LIN {X 0,Y 247.76,Z 536.952,A -85,B 0,C 180,E1 -18799.376,E2 -18799.376} C_VEL
LIN {X 0,Y 247.256,Z 541.833,A -85,B 0,C 180,E1 -18801.831,E2 -18801.831} C_VEL
LIN {X 0,Y 246.931,Z 545.565,A -85,B 0,C 180,E1 -18804.284,E2 -18804.284} C_VEL
LIN {X 0,Y 246.895,Z 548.265,A -85,B 0,C 180,E1 -18806.738,E2 -18806.738} C_VEL
LIN {X 0,Y 246.957,Z 549.533,A -85,B 0,C 180,E1 -18808.37,E2 -18808.37} C_VEL
LIN {X 0,Y 246.985,Z 550.397,A -85,B 0,C 180,E1 -18810.001,E2 -18810.001} C_VEL
LIN {X 0,Y 246.925,Z 550.819,A -85,B 0,C 180,E1 -18811.632,E2 -18811.632} C_VEL
LIN {X 0,Y 246.882,Z 550.489,A -85,B 0,C 180,E1 -18814.9,E2 -18814.9} C_VEL
LIN {X 0,Y 247.022,Z 549.754,A -85,B 0,C 180,E1 -18816.536,E2 -18816.536} C_VEL
LIN {X 0,Y 247.296,Z 548.597,A -85,B 0,C 180,E1 -18818.17,E2 -18818.17} C_VEL
LIN {X 0,Y 247.735,Z 547.02,A -85,B 0,C 180,E1 -18819.801,E2 -18819.801} C_VEL
LIN {X 0,Y 248.65,Z 543.875,A -85,B 0,C 180,E1 -18822.24,E2 -18822.24} C_VEL
LIN {X 0,Y 249.943,Z 539.694,A -85,B 0,C 180,E1 -18824.66,E2 -18824.66} C_VEL
LIN {X 0,Y 252.206,Z 533.352,A -85,B 0,C 180,E1 -18827.432,E2 -18827.432} C_VEL
LIN {X 0,Y 254.652,Z 525.61,A -85,B 0,C 180,E1 -18830.038,E2 -18830.038} C_VEL
LIN {X 0,Y 256.959,Z 517.893,A -85,B 0,C 180,E1 -18832.092,E2 -18832.092} C_VEL
LIN {X 0,Y 259.561,Z 509.116,A -85,B 0,C 180,E1 -18833.964,E2 -18833.964} C_VEL
LIN {X 0,Y 262.449,Z 498.336,A -85,B 0,C 180,E1 -18835.796,E2 -18835.796} C_VEL
LIN {X 0,Y 264.991,Z 487.513,A -85,B 0,C 180,E1 -18837.227,E2 -18837.227} C_VEL
LIN {X 0,Y 267.415,Z 475.396,A -85,B 0,C 180,E1 -18838.448,E2 -18838.448} C_VEL
LIN {X 0,Y 269.44,Z 462.72,A -85,B 0,C 180,E1 -18839.388,E2 -18839.388} C_VEL
LIN {X 0,Y 270.794,Z 450.762,A -85,B 0,C 180,E1 -18839.998,E2 -18839.998} C_VEL
LIN {X 0,Y 271.642,Z 434.886,A -85,B 0,C 180,E1 -18840.499,E2 -18840.499} C_VEL
LIN {X 0,Y 273.321,Z 390.073,A -85,B 0,C 180,E1 -18841.676,E2 -18841.676} C_VEL
LIN {X 0,Y 270.28,Z 372.943,A -85,B 0,C 180,E1 -18842.701,E2 -18842.701} C_VEL
LIN {X 0,Y 265.11,Z 361.26,A -85,B 0,C 180,E1 -18843.938,E2 -18843.938} C_VEL
LIN {X 0,Y 257.601,Z 346.459,A -85,B 0,C 180,E1 -18845.793,E2 -18845.793} C_VEL
LIN {X 0,Y 254.306,Z 340.666,A -85,B 0,C 180,E1 -18846.634,E2 -18846.634} C_VEL
LIN {X 0,Y 252.61,Z 337.257,A -85,B 0,C 180,E1 -18847.12,E2 -18847.12} C_VEL
LIN {X 0,Y 250.483,Z 329.649,A -85,B 0,C 180,E1 -18850.751,E2 -18850.751} C_VEL
LIN {X 0,Y 249.027,Z 324.462,A -85,B 0,C 180,E1 -18853.427,E2 -18853.427} C_VEL
LIN {X 0,Y 249.012,Z 324.468,A -85,B 0,C 180,E1 -18857.362,E2 -18857.362} C_VEL
LIN {X 0,Y 249.027,Z 324.458,A -85,B 0,C 180,E1 -18861.62,E2 -18861.62} C_VEL
LIN {X 0,Y 249.045,Z 324.46,A -85,B 0,C 180,E1 -18865.64,E2 -18865.64} C_VEL
LIN {X 0,Y 249.005,Z 324.468,A -85,B 0,C 180,E1 -18869.467,E2 -18869.467} C_VEL
LIN {X 0,Y 249.04,Z 324.464,A -85,B 0,C 180,E1 -18873.159,E2 -18873.159} C_VEL
LIN {X 0,Y 249.128,Z 324.445,A -85,B 0,C 180,E1 -18874.966,E2 -18874.966} C_VEL
LIN {X 0,Y 249.092,Z 324.45,A -85,B 0,C 180,E1 -18878.605,E2 -18878.605} C_VEL
LIN {X 0,Y 249.179,Z 324.436,A -85,B 0,C 180,E1 -18883.618,E2 -18883.618} C_VEL
LIN {X 0,Y 249.237,Z 324.432,A -85,B 0,C 180,E1 -18888.616,E2 -18888.616} C_VEL
LIN {X 0,Y 249.448,Z 324.398,A -85,B 0,C 180,E1 -18891.902,E2 -18891.902} C_VEL
LIN {X 0,Y 249.281,Z 324.423,A -85,B 0,C 180,E1 -18895.148,E2 -18895.148} C_VEL
LIN {X 0,Y 249.666,Z 324.381,A -85,B 0,C 180,E1 -18898.387,E2 -18898.387} C_VEL
LIN {X 0,Y 249.673,Z 324.375,A -85,B 0,C 180,E1 -18901.613,E2 -18901.613} C_VEL
LIN {X 0,Y 249.432,Z 324.41,A -85,B 0,C 180,E1 -18906.577,E2 -18906.577} C_VEL
LIN {X 0,Y 249.346,Z 324.415,A -85,B 0,C 180,E1 -18909.737,E2 -18909.737} C_VEL
LIN {X 0,Y 249.185,Z 324.441,A -85,B 0,C 180,E1 -18914.705,E2 -18914.705} C_VEL
LIN {X 0,Y 249.116,Z 324.444,A -85,B 0,C 180,E1 -18918.08,E2 -18918.08} C_VEL
LIN {X 0,Y 249.084,Z 324.447,A -85,B 0,C 180,E1 -18921.519,E2 -18921.519} C_VEL
LIN {X 0,Y 249.108,Z 324.445,A -85,B 0,C 180,E1 -18925.469,E2 -18925.469} C_VEL
LIN {X 0,Y 249.045,Z 324.454,A -85,B 0,C 180,E1 -18928.976,E2 -18928.976} C_VEL
LIN {X 0,Y 249.031,Z 324.459,A -85,B 0,C 180,E1 -18932.426,E2 -18932.426} C_VEL
LIN {X 0,Y 249.057,Z 324.462,A -85,B 0,C 180,E1 -18936.341,E2 -18936.341} C_VEL
LIN {X 0,Y 249.034,Z 324.542,A -85,B 0,C 180,E1 -18940.134,E2 -18940.134} C_VEL
LIN {X 0,Y 249.7,Z 326.855,A -85,B 0,C 180,E1 -18941.342,E2 -18941.342} C_VEL
LIN {X 0,Y 251.823,Z 330.474,A -85,B 0,C 180,E1 -18941.918,E2 -18941.918} C_VEL
LIN {X 0,Y 258.717,Z 342.019,A -85,B 0,C 180,E1 -18943.683,E2 -18943.683} C_VEL
LIN {X 0,Y 265.785,Z 354.94,A -85,B 0,C 180,E1 -18945.389,E2 -18945.389} C_VEL
LIN {X 0,Y 272.354,Z 368.856,A -85,B 0,C 180,E1 -18946.92,E2 -18946.92} C_VEL
LIN {X 0,Y 274.083,Z 372.882,A -85,B 0,C 180,E1 -18947.317,E2 -18947.317} C_VEL
LIN {X 0,Y 271.457,Z 434.189,A -85,B 0,C 180,E1 -18948.929,E2 -18948.929} C_VEL
LIN {X 0,Y 270.158,Z 447.569,A -85,B 0,C 180,E1 -18949.553,E2 -18949.553} C_VEL
LIN {X 0,Y 268.442,Z 460.42,A -85,B 0,C 180,E1 -18950.466,E2 -18950.466} C_VEL
LIN {X 0,Y 266.639,Z 470.957,A -85,B 0,C 180,E1 -18951.485,E2 -18951.485} C_VEL
LIN {X 0,Y 264.44,Z 481.999,A -85,B 0,C 180,E1 -18952.875,E2 -18952.875} C_VEL
LIN {X 0,Y 261.843,Z 492.45,A -85,B 0,C 180,E1 -18954.519,E2 -18954.519} C_VEL
LIN {X 0,Y 259.378,Z 501.292,A -85,B 0,C 180,E1 -18956.257,E2 -18956.257} C_VEL
LIN {X 0,Y 257.008,Z 508.957,A -85,B 0,C 180,E1 -18958.107,E2 -18958.107} C_VEL
LIN {X 0,Y 254.704,Z 516.048,A -85,B 0,C 180,E1 -18960.219,E2 -18960.219} C_VEL
LIN {X 0,Y 252.49,Z 522.427,A -85,B 0,C 180,E1 -18962.608,E2 -18962.608} C_VEL
LIN {X 0,Y 250.658,Z 527.635,A -85,B 0,C 180,E1 -18965.128,E2 -18965.128} C_VEL
LIN {X 0,Y 249.218,Z 531.546,A -85,B 0,C 180,E1 -18967.622,E2 -18967.622} C_VEL
LIN {X 0,Y 248.163,Z 534.375,A -85,B 0,C 180,E1 -18970.132,E2 -18970.132} C_VEL
LIN {X 0,Y 247.596,Z 535.692,A -85,B 0,C 180,E1 -18971.805,E2 -18971.805} C_VEL
LIN {X 0,Y 247.213,Z 536.602,A -85,B 0,C 180,E1 -18973.483,E2 -18973.483} C_VEL
LIN {X 0,Y 247.008,Z 537.095,A -85,B 0,C 180,E1 -18975.329,E2 -18975.329} C_VEL
LIN {X 0,Y 246.707,Z 536.789,A -85,B 0,C 180,E1 -18978.496,E2 -18978.496} C_VEL
LIN {X 0,Y 246.697,Z 536.057,A -85,B 0,C 180,E1 -18980.157,E2 -18980.157} C_VEL
LIN {X 0,Y 246.776,Z 534.889,A -85,B 0,C 180,E1 -18981.812,E2 -18981.812} C_VEL
LIN {X 0,Y 247.107,Z 532.038,A -85,B 0,C 180,E1 -18984.532,E2 -18984.532} C_VEL
LIN {X 0,Y 247.482,Z 528.833,A -85,B 0,C 180,E1 -18986.743,E2 -18986.743} C_VEL
LIN {X 0,Y 248.065,Z 524.207,A -85,B 0,C 180,E1 -18989.187,E2 -18989.187} C_VEL
LIN {X 0,Y 249.055,Z 517.233,A -85,B 0,C 180,E1 -18992.02,E2 -18992.02} C_VEL
LIN {X 0,Y 250.459,Z 509.671,A -85,B 0,C 180,E1 -18994.424,E2 -18994.424} C_VEL
LIN {X 0,Y 251.668,Z 501.97,A -85,B 0,C 180,E1 -18996.412,E2 -18996.412} C_VEL
LIN {X 0,Y 253.45,Z 491.482,A -85,B 0,C 180,E1 -18998.57,E2 -18998.57} C_VEL
LIN {X 0,Y 255.305,Z 480.769,A -85,B 0,C 180,E1 -19000.306,E2 -19000.306} C_VEL
LIN {X 0,Y 256.637,Z 470.452,A -85,B 0,C 180,E1 -19001.651,E2 -19001.651} C_VEL
LIN {X 0,Y 257.901,Z 458.119,A -85,B 0,C 180,E1 -19002.891,E2 -19002.891} C_VEL
LIN {X 0,Y 258.968,Z 445.126,A -85,B 0,C 180,E1 -19003.836,E2 -19003.836} C_VEL
LIN {X 0,Y 259.706,Z 432.827,A -85,B 0,C 180,E1 -19004.425,E2 -19004.425} C_VEL
LIN {X 0,Y 261.92,Z 361.963,A -85,B 0,C 180,E1 -19006.338,E2 -19006.338} C_VEL
LIN {X 0,Y 260.684,Z 355.255,A -85,B 0,C 180,E1 -19006.654,E2 -19006.654} C_VEL
LIN {X 0,Y 254.665,Z 338.73,A -85,B 0,C 180,E1 -19007.751,E2 -19007.751} C_VEL
LIN {X 0,Y 249.434,Z 325.955,A -85,B 0,C 180,E1 -19008.725,E2 -19008.725} C_VEL
LIN {X 0,Y 249.101,Z 324.46,A -85,B 0,C 180,E1 -19009.359,E2 -19009.359} C_VEL
LIN {X 0,Y 249.012,Z 324.466,A -85,B 0,C 180,E1 -19013.273,E2 -19013.273} C_VEL
LIN {X 0,Y 249.014,Z 324.466,A -85,B 0,C 180,E1 -19016.843,E2 -19016.843} C_VEL
LIN {X 0,Y 248.992,Z 324.468,A -85,B 0,C 180,E1 -19020.533,E2 -19020.533} C_VEL
LIN {X 0,Y 249.041,Z 324.463,A -85,B 0,C 180,E1 -19024.359,E2 -19024.359} C_VEL
LIN {X 0,Y 249.02,Z 324.466,A -85,B 0,C 180,E1 -19028.38,E2 -19028.38} C_VEL
LIN {X 0,Y 248.967,Z 324.472,A -85,B 0,C 180,E1 -19032.781,E2 -19032.781} C_VEL
LIN {X 0,Y 248.975,Z 324.463,A -85,B 0,C 180,E1 -19037.353,E2 -19037.353} C_VEL
LIN {X 0,Y 249.036,Z 324.459,A -85,B 0,C 180,E1 -19042.2,E2 -19042.2} C_VEL
LIN {X 0,Y 249.038,Z 324.454,A -85,B 0,C 180,E1 -19045.638,E2 -19045.638} C_VEL
LIN {X 0,Y 248.988,Z 324.47,A -85,B 0,C 180,E1 -19049.464,E2 -19049.464} C_VEL
LIN {X 0,Y 249.007,Z 324.457,A -85,B 0,C 180,E1 -19053.154,E2 -19053.154} C_VEL
LIN {X 0,Y 249,Z 324.462,A -85,B 0,C 180,E1 -19056.724,E2 -19056.724} C_VEL
LIN {X 0,Y 249.035,Z 324.462,A -85,B 0,C 180,E1 -19060.205,E2 -19060.205} C_VEL
LIN {X 0,Y 249.151,Z 324.437,A -85,B 0,C 180,E1 -19063.615,E2 -19063.615} C_VEL
LIN {X 0,Y 249.207,Z 324.44,A -85,B 0,C 180,E1 -19068.614,E2 -19068.614} C_VEL
LIN {X 0,Y 249.395,Z 324.418,A -85,B 0,C 180,E1 -19071.9,E2 -19071.9} C_VEL
LIN {X 0,Y 249.256,Z 324.418,A -85,B 0,C 180,E1 -19075.147,E2 -19075.147} C_VEL
LIN {X 0,Y 249.65,Z 324.384,A -85,B 0,C 180,E1 -19078.387,E2 -19078.387} C_VEL
LIN {X 0,Y 249.653,Z 324.384,A -85,B 0,C 180,E1 -19081.613,E2 -19081.613} C_VEL
LIN {X 0,Y 249.271,Z 324.42,A -85,B 0,C 180,E1 -19084.446,E2 -19084.446} C_VEL
LIN {X 0,Y 248.563,Z 324.509,A -85,B 0,C 180,E1 -19085.796,E2 -19085.796} C_VEL
LIN {X 0,Y 245.684,Z 324.873,A -85,B 0,C 180,E1 -19087.997,E2 -19087.997} C_VEL
LIN {X 0,Y 243.266,Z 325.18,A -85,B 0,C 180,E1 -19089.79,E2 -19089.79} C_VEL
LIN {X 0,Y 242.238,Z 325.309,A -85,B 0,C 180,E1 -19091.181,E2 -19091.181} C_VEL
LIN {X 0,Y 242.157,Z 325.318,A -85,B 0,C 180,E1 -19091.652,E2 -19091.652} C_VEL
LIN {X 0,Y 242.127,Z 325.31,A -85,B 0,C 180,E1 -19095.143,E2 -19095.143} C_VEL
LIN {X 0,Y 242.039,Z 325.332,A -85,B 0,C 180,E1 -19098.627,E2 -19098.627} C_VEL
LIN {X 0,Y 241.997,Z 325.337,A -85,B 0,C 180,E1 -19102.181,E2 -19102.181} C_VEL
LIN {X 0,Y 242.06,Z 325.331,A -85,B 0,C 180,E1 -19105.839,E2 -19105.839} C_VEL
LIN {X 0,Y 241.997,Z 325.34,A -85,B 0,C 180,E1 -19109.584,E2 -19109.584} C_VEL
LIN {X 0,Y 241.974,Z 325.341,A -85,B 0,C 180,E1 -19113.493,E2 -19113.493} C_VEL
LIN {X 0,Y 241.978,Z 325.342,A -85,B 0,C 180,E1 -19117.584,E2 -19117.584} C_VEL
LIN {X 0,Y 241.922,Z 325.341,A -85,B 0,C 180,E1 -19121.926,E2 -19121.926} C_VEL
LIN {X 0,Y 241.928,Z 325.348,A -85,B 0,C 180,E1 -19126.573,E2 -19126.573} C_VEL
LIN {X 0,Y 241.953,Z 325.346,A -85,B 0,C 180,E1 -19130.282,E2 -19130.282} C_VEL
LIN {X 0,Y 242.022,Z 325.376,A -85,B 0,C 180,E1 -19134.752,E2 -19134.752} C_VEL
LIN {X 0,Y 244.291,Z 335.575,A -85,B 0,C 180,E1 -19138.814,E2 -19138.814} C_VEL
LIN {X 0,Y 244.805,Z 338.084,A -85,B 0,C 180,E1 -19139.777,E2 -19139.777} C_VEL
LIN {X 0,Y 250.658,Z 354.288,A -85,B 0,C 180,E1 -19140.948,E2 -19140.948} C_VEL
LIN {X 0,Y 254.821,Z 387.155,A -85,B 0,C 180,E1 -19142.371,E2 -19142.371} C_VEL
LIN {X 0,Y 253.039,Z 447.068,A -85,B 0,C 180,E1 -19144.06,E2 -19144.06} C_VEL
LIN {X 0,Y 252.03,Z 460.992,A -85,B 0,C 180,E1 -19144.78,E2 -19144.78} C_VEL
LIN {X 0,Y 250.73,Z 472.9,A -85,B 0,C 180,E1 -19145.69,E2 -19145.69} C_VEL
LIN {X 0,Y 249.168,Z 484.968,A -85,B 0,C 180,E1 -19146.963,E2 -19146.963} C_VEL
LIN {X 0,Y 247.315,Z 496.492,A -85,B 0,C 180,E1 -19148.54,E2 -19148.54} C_VEL
LIN {X 0,Y 245.783,Z 505.922,A -85,B 0,C 180,E1 -19150.173,E2 -19150.173} C_VEL
LIN {X 0,Y 244.408,Z 514.497,A -85,B 0,C 180,E1 -19151.995,E2 -19151.995} C_VEL
LIN {X 0,Y 242.999,Z 522.478,A -85,B 0,C 180,E1 -19154.054,E2 -19154.054} C_VEL
LIN {X 0,Y 241.62,Z 530.25,A -85,B 0,C 180,E1 -19156.546,E2 -19156.546} C_VEL
LIN {X 0,Y 240.765,Z 536.487,A -85,B 0,C 180,E1 -19159.064,E2 -19159.064} C_VEL
LIN {X 0,Y 240.199,Z 541.424,A -85,B 0,C 180,E1 -19161.589,E2 -19161.589} C_VEL
LIN {X 0,Y 239.859,Z 545.21,A -85,B 0,C 180,E1 -19164.115,E2 -19164.115} C_VEL
LIN {X 0,Y 239.797,Z 547.96,A -85,B 0,C 180,E1 -19166.641,E2 -19166.641} C_VEL
LIN {X 0,Y 239.865,Z 549.252,A -85,B 0,C 180,E1 -19168.322,E2 -19168.322} C_VEL
LIN {X 0,Y 239.915,Z 550.143,A -85,B 0,C 180,E1 -19170.001,E2 -19170.001} C_VEL
LIN {X 0,Y 239.834,Z 550.609,A -85,B 0,C 180,E1 -19171.68,E2 -19171.68} C_VEL
LIN {X 0,Y 239.801,Z 550.325,A -85,B 0,C 180,E1 -19175.045,E2 -19175.045} C_VEL
LIN {X 0,Y 239.962,Z 549.613,A -85,B 0,C 180,E1 -19176.729,E2 -19176.729} C_VEL
LIN {X 0,Y 240.245,Z 548.502,A -85,B 0,C 180,E1 -19178.412,E2 -19178.412} C_VEL
LIN {X 0,Y 240.717,Z 546.951,A -85,B 0,C 180,E1 -19180.09,E2 -19180.09} C_VEL
LIN {X 0,Y 241.698,Z 543.859,A -85,B 0,C 180,E1 -19182.598,E2 -19182.598} C_VEL
LIN {X 0,Y 243.077,Z 539.735,A -85,B 0,C 180,E1 -19185.084,E2 -19185.084} C_VEL
LIN {X 0,Y 245.438,Z 533.455,A -85,B 0,C 180,E1 -19187.929,E2 -19187.929} C_VEL
LIN {X 0,Y 247.871,Z 526.214,A -85,B 0,C 180,E1 -19190.477,E2 -19190.477} C_VEL
LIN {X 0,Y 250.401,Z 518.185,A -85,B 0,C 180,E1 -19192.702,E2 -19192.702} C_VEL
LIN {X 0,Y 253.116,Z 509.504,A -85,B 0,C 180,E1 -19194.614,E2 -19194.614} C_VEL
LIN {X 0,Y 256.107,Z 498.843,A -85,B 0,C 180,E1 -19196.484,E2 -19196.484} C_VEL
LIN {X 0,Y 258.73,Z 488.244,A -85,B 0,C 180,E1 -19197.942,E2 -19197.942} C_VEL
LIN {X 0,Y 261.238,Z 476.392,A -85,B 0,C 180,E1 -19199.185,E2 -19199.185} C_VEL
LIN {X 0,Y 263.308,Z 464.088,A -85,B 0,C 180,E1 -19200.142,E2 -19200.142} C_VEL
LIN {X 0,Y 264.831,Z 451.657,A -85,B 0,C 180,E1 -19200.821,E2 -19200.821} C_VEL
LIN {X 0,Y 265.732,Z 437.784,A -85,B 0,C 180,E1 -19201.288,E2 -19201.288} C_VEL
LIN {X 0,Y 267.573,Z 391.152,A -85,B 0,C 180,E1 -19202.532,E2 -19202.532} C_VEL
LIN {X 0,Y 264.877,Z 375.804,A -85,B 0,C 180,E1 -19203.484,E2 -19203.484} C_VEL
LIN {X 0,Y 258.917,Z 362.515,A -85,B 0,C 180,E1 -19204.98,E2 -19204.98} C_VEL
LIN {X 0,Y 252.722,Z 350.413,A -85,B 0,C 180,E1 -19206.583,E2 -19206.583} C_VEL
LIN {X 0,Y 247.642,Z 341.288,A -85,B 0,C 180,E1 -19207.96,E2 -19207.96} C_VEL
LIN {X 0,Y 245.361,Z 337.151,A -85,B 0,C 180,E1 -19208.61,E2 -19208.61} C_VEL
LIN {X 0,Y 243.084,Z 329.298,A -85,B 0,C 180,E1 -19212.569,E2 -19212.569} C_VEL
LIN {X 0,Y 241.947,Z 325.349,A -85,B 0,C 180,E1 -19214.816,E2 -19214.816} C_VEL
LIN {X 0,Y 241.934,Z 325.344,A -85,B 0,C 180,E1 -19219.051,E2 -19219.051} C_VEL
LIN {X 0,Y 241.99,Z 325.337,A -85,B 0,C 180,E1 -19222.418,E2 -19222.418} C_VEL
LIN {X 0,Y 241.982,Z 325.344,A -85,B 0,C 180,E1 -19226.508,E2 -19226.508} C_VEL
LIN {X 0,Y 241.98,Z 325.339,A -85,B 0,C 180,E1 -19230.613,E2 -19230.613} C_VEL
LIN {X 0,Y 242.035,Z 325.334,A -85,B 0,C 180,E1 -19234.179,E2 -19234.179} C_VEL
LIN {X 0,Y 242.025,Z 325.332,A -85,B 0,C 180,E1 -19238.316,E2 -19238.316} C_VEL
LIN {X 0,Y 242.118,Z 325.315,A -85,B 0,C 180,E1 -19243.317,E2 -19243.317} C_VEL
LIN {X 0,Y 242.171,Z 325.309,A -85,B 0,C 180,E1 -19248.279,E2 -19248.279} C_VEL
LIN {X 0,Y 242.396,Z 325.276,A -85,B 0,C 180,E1 -19251.665,E2 -19251.665} C_VEL
LIN {X 0,Y 242.418,Z 325.281,A -85,B 0,C 180,E1 -19253.341,E2 -19253.341} C_VEL
LIN {X 0,Y 242.626,Z 325.258,A -85,B 0,C 180,E1 -19258.34,E2 -19258.34} C_VEL
LIN {X 0,Y 242.633,Z 325.252,A -85,B 0,C 180,E1 -19261.66,E2 -19261.66} C_VEL
LIN {X 0,Y 242.41,Z 325.287,A -85,B 0,C 180,E1 -19266.66,E2 -19266.66} C_VEL
LIN {X 0,Y 242.271,Z 325.298,A -85,B 0,C 180,E1 -19270.024,E2 -19270.024} C_VEL
LIN {X 0,Y 242.142,Z 325.323,A -85,B 0,C 180,E1 -19275.143,E2 -19275.143} C_VEL
LIN {X 0,Y 242.054,Z 325.327,A -85,B 0,C 180,E1 -19278.626,E2 -19278.626} C_VEL
LIN {X 0,Y 242.007,Z 325.33,A -85,B 0,C 180,E1 -19282.181,E2 -19282.181} C_VEL
LIN {X 0,Y 242.036,Z 325.327,A -85,B 0,C 180,E1 -19285.821,E2 -19285.821} C_VEL
LIN {X 0,Y 241.974,Z 325.339,A -85,B 0,C 180,E1 -19289.588,E2 -19289.588} C_VEL
LIN {X 0,Y 241.984,Z 325.341,A -85,B 0,C 180,E1 -19293.493,E2 -19293.493} C_VEL
LIN {X 0,Y 241.997,Z 325.337,A -85,B 0,C 180,E1 -19297.581,E2 -19297.581} C_VEL
LIN {X 0,Y 242.007,Z 325.528,A -85,B 0,C 180,E1 -19298.885,E2 -19298.885} C_VEL
LIN {X 0,Y 242.52,Z 327.239,A -85,B 0,C 180,E1 -19299.787,E2 -19299.787} C_VEL
LIN {X 0,Y 244.822,Z 331.105,A -85,B 0,C 180,E1 -19300.459,E2 -19300.459} C_VEL
LIN {X 0,Y 249.296,Z 338.205,A -85,B 0,C 180,E1 -19301.694,E2 -19301.694} C_VEL
LIN {X 0,Y 256.585,Z 350.68,A -85,B 0,C 180,E1 -19303.595,E2 -19303.595} C_VEL
LIN {X 0,Y 264.622,Z 366.569,A -85,B 0,C 180,E1 -19305.586,E2 -19305.586} C_VEL
LIN {X 0,Y 268.228,Z 374.835,A -85,B 0,C 180,E1 -19306.461,E2 -19306.461} C_VEL
LIN {X 0,Y 265.699,Z 433.719,A -85,B 0,C 180,E1 -19308.041,E2 -19308.041} C_VEL
LIN {X 0,Y 264.359,Z 447.177,A -85,B 0,C 180,E1 -19308.663,E2 -19308.663} C_VEL
LIN {X 0,Y 262.678,Z 459.629,A -85,B 0,C 180,E1 -19309.547,E2 -19309.547} C_VEL
LIN {X 0,Y 260.957,Z 469.495,A -85,B 0,C 180,E1 -19310.486,E2 -19310.486} C_VEL
LIN {X 0,Y 258.627,Z 480.973,A -85,B 0,C 180,E1 -19311.898,E2 -19311.898} C_VEL
LIN {X 0,Y 255.901,Z 491.616,A -85,B 0,C 180,E1 -19313.565,E2 -19313.565} C_VEL
LIN {X 0,Y 253.3,Z 500.63,A -85,B 0,C 180,E1 -19315.333,E2 -19315.333} C_VEL
LIN {X 0,Y 250.827,Z 508.371,A -85,B 0,C 180,E1 -19317.203,E2 -19317.203} C_VEL
LIN {X 0,Y 248.334,Z 515.653,A -85,B 0,C 180,E1 -19319.374,E2 -19319.374} C_VEL
LIN {X 0,Y 245.881,Z 522.479,A -85,B 0,C 180,E1 -19321.952,E2 -19321.952} C_VEL
LIN {X 0,Y 244.014,Z 527.492,A -85,B 0,C 180,E1 -19324.403,E2 -19324.403} C_VEL
LIN {X 0,Y 242.431,Z 531.489,A -85,B 0,C 180,E1 -19326.96,E2 -19326.96} C_VEL
LIN {X 0,Y 241.281,Z 534.4,A -85,B 0,C 180,E1 -19329.54,E2 -19329.54} C_VEL
LIN {X 0,Y 240.65,Z 535.757,A -85,B 0,C 180,E1 -19331.261,E2 -19331.261} C_VEL
LIN {X 0,Y 240.218,Z 536.706,A -85,B 0,C 180,E1 -19332.987,E2 -19332.987} C_VEL
LIN {X 0,Y 239.954,Z 537.299,A -85,B 0,C 180,E1 -19335.138,E2 -19335.138} C_VEL
LIN {X 0,Y 239.617,Z 537.049,A -85,B 0,C 180,E1 -19338.151,E2 -19338.151} C_VEL
LIN {X 0,Y 239.604,Z 536.355,A -85,B 0,C 180,E1 -19339.863,E2 -19339.863} C_VEL
LIN {X 0,Y 239.654,Z 535.261,A -85,B 0,C 180,E1 -19341.567,E2 -19341.567} C_VEL
LIN {X 0,Y 240.028,Z 532.224,A -85,B 0,C 180,E1 -19344.581,E2 -19344.581} C_VEL
LIN {X 0,Y 240.495,Z 527.947,A -85,B 0,C 180,E1 -19347.486,E2 -19347.486} C_VEL
LIN {X 0,Y 241.204,Z 523.028,A -85,B 0,C 180,E1 -19349.999,E2 -19349.999} C_VEL
LIN {X 0,Y 242.166,Z 516.848,A -85,B 0,C 180,E1 -19352.494,E2 -19352.494} C_VEL
LIN {X 0,Y 243.629,Z 509.127,A -85,B 0,C 180,E1 -19354.963,E2 -19354.963} C_VEL
LIN {X 0,Y 245.251,Z 499.474,A -85,B 0,C 180,E1 -19357.408,E2 -19357.408} C_VEL
LIN {X 0,Y 246.872,Z 490.551,A -85,B 0,C 180,E1 -19359.213,E2 -19359.213} C_VEL
LIN {X 0,Y 248.772,Z 479.553,A -85,B 0,C 180,E1 -19360.992,E2 -19360.992} C_VEL
LIN {X 0,Y 250.126,Z 468.842,A -85,B 0,C 180,E1 -19362.37,E2 -19362.37} C_VEL
LIN {X 0,Y 251.471,Z 455.955,A -85,B 0,C 180,E1 -19363.638,E2 -19363.638} C_VEL
LIN {X 0,Y 252.484,Z 443.567,A -85,B 0,C 180,E1 -19364.507,E2 -19364.507} C_VEL
LIN {X 0,Y 253.206,Z 430.694,A -85,B 0,C 180,E1 -19365.081,E2 -19365.081} C_VEL
LIN {X 0,Y 255.446,Z 363.045,A -85,B 0,C 180,E1 -19366.931,E2 -19366.931} C_VEL
LIN {X 0,Y 254.351,Z 357.299,A -85,B 0,C 180,E1 -19367.215,E2 -19367.215} C_VEL
LIN {X 0,Y 248.417,Z 341.025,A -85,B 0,C 180,E1 -19368.339,E2 -19368.339} C_VEL
LIN {X 0,Y 242.191,Z 326.126,A -85,B 0,C 180,E1 -19369.558,E2 -19369.558} C_VEL
LIN {X 0,Y 242.015,Z 325.341,A -85,B 0,C 180,E1 -19369.95,E2 -19369.95} C_VEL
LIN {X 0,Y 241.985,Z 325.344,A -85,B 0,C 180,E1 -19373.99,E2 -19373.99} C_VEL
LIN {X 0,Y 241.951,Z 325.345,A -85,B 0,C 180,E1 -19377.693,E2 -19377.693} C_VEL
LIN {X 0,Y 241.947,Z 325.344,A -85,B 0,C 180,E1 -19381.522,E2 -19381.522} C_VEL
LIN {X 0,Y 241.976,Z 325.34,A -85,B 0,C 180,E1 -19385.586,E2 -19385.586} C_VEL
LIN {X 0,Y 241.937,Z 325.344,A -85,B 0,C 180,E1 -19389.721,E2 -19389.721} C_VEL
LIN {X 0,Y 241.893,Z 325.352,A -85,B 0,C 180,E1 -19394.209,E2 -19394.209} C_VEL
LIN {X 0,Y 241.904,Z 325.343,A -85,B 0,C 180,E1 -19398.07,E2 -19398.07} C_VEL
LIN {X 0,Y 241.978,Z 325.339,A -85,B 0,C 180,E1 -19402.415,E2 -19402.415} C_VEL
LIN {X 0,Y 241.973,Z 325.334,A -85,B 0,C 180,E1 -19406.506,E2 -19406.506} C_VEL
LIN {X 0,Y 241.964,Z 325.341,A -85,B 0,C 180,E1 -19410.614,E2 -19410.614} C_VEL
LIN {X 0,Y 241.99,Z 325.325,A -85,B 0,C 180,E1 -19414.196,E2 -19414.196} C_VEL
LIN {X 0,Y 241.979,Z 325.341,A -85,B 0,C 180,E1 -19418.337,E2 -19418.337} C_VEL
LIN {X 0,Y 242.099,Z 325.317,A -85,B 0,C 180,E1 -19423.324,E2 -19423.324} C_VEL
LIN {X 0,Y 242.141,Z 325.322,A -85,B 0,C 180,E1 -19428.277,E2 -19428.277} C_VEL
LIN {X 0,Y 242.351,Z 325.295,A -85,B 0,C 180,E1 -19431.663,E2 -19431.663} C_VEL
LIN {X 0,Y 242.384,Z 325.284,A -85,B 0,C 180,E1 -19433.339,E2 -19433.339} C_VEL
LIN {X 0,Y 242.61,Z 325.26,A -85,B 0,C 180,E1 -19438.34,E2 -19438.34} C_VEL
LIN {X 0,Y 242.613,Z 325.261,A -85,B 0,C 180,E1 -19441.66,E2 -19441.66} C_VEL
LIN {X 0,Y 242.398,Z 325.277,A -85,B 0,C 180,E1 -19446.66,E2 -19446.66} C_VEL
LIN {X 0,Y 242.254,Z 325.306,A -85,B 0,C 180,E1 -19450.024,E2 -19450.024} C_VEL
LIN {X 0,Y 242.157,Z 325.318,A -85,B 0,C 180,E1 -19451.652,E2 -19451.652} C_VEL
LIN {X 0,Y 241.474,Z 325.408,A -85,B 0,C 180,E1 -19453.041,E2 -19453.041} C_VEL
LIN {X 0,Y 238.543,Z 325.767,A -85,B 0,C 180,E1 -19455.302,E2 -19455.302} C_VEL
LIN {X 0,Y 236.071,Z 326.07,A -85,B 0,C 180,E1 -19457.145,E2 -19457.145} C_VEL
LIN {X 0,Y 235.041,Z 326.203,A -85,B 0,C 180,E1 -19458.578,E2 -19458.578} C_VEL
LIN {X 0,Y 234.974,Z 326.215,A -85,B 0,C 180,E1 -19459.064,E2 -19459.064} C_VEL
LIN {X 0,Y 234.944,Z 326.215,A -85,B 0,C 180,E1 -19462.884,E2 -19462.884} C_VEL
LIN {X 0,Y 234.957,Z 326.216,A -85,B 0,C 180,E1 -19466.659,E2 -19466.659} C_VEL
LIN {X 0,Y 234.915,Z 326.22,A -85,B 0,C 180,E1 -19470.57,E2 -19470.57} C_VEL
LIN {X 0,Y 234.92,Z 326.22,A -85,B 0,C 180,E1 -19474.64,E2 -19474.64} C_VEL
LIN {X 0,Y 234.906,Z 326.223,A -85,B 0,C 180,E1 -19478.936,E2 -19478.936} C_VEL
LIN {X 0,Y 234.873,Z 326.223,A -85,B 0,C 180,E1 -19483.489,E2 -19483.489} C_VEL
LIN {X 0,Y 234.88,Z 326.226,A -85,B 0,C 180,E1 -19486.515,E2 -19486.515} C_VEL
LIN {X 0,Y 234.916,Z 326.223,A -85,B 0,C 180,E1 -19491.08,E2 -19491.08} C_VEL
LIN {X 0,Y 234.976,Z 326.324,A -85,B 0,C 180,E1 -19494.183,E2 -19494.183} C_VEL
LIN {X 0,Y 237.092,Z 335.887,A -85,B 0,C 180,E1 -19498.131,E2 -19498.131} C_VEL
LIN {X 0,Y 237.606,Z 338.201,A -85,B 0,C 180,E1 -19498.97,E2 -19498.97} C_VEL
LIN {X 0,Y 244.375,Z 356.437,A -85,B 0,C 180,E1 -19500.343,E2 -19500.343} C_VEL
LIN {X 0,Y 248.2,Z 386.732,A -85,B 0,C 180,E1 -19501.704,E2 -19501.704} C_VEL
LIN {X 0,Y 246.5,Z 446.385,A -85,B 0,C 180,E1 -19503.433,E2 -19503.433} C_VEL
LIN {X 0,Y 245.52,Z 459.7,A -85,B 0,C 180,E1 -19504.119,E2 -19504.119} C_VEL
LIN {X 0,Y 244.107,Z 472.463,A -85,B 0,C 180,E1 -19505.1,E2 -19505.1} C_VEL
LIN {X 0,Y 242.625,Z 483.805,A -85,B 0,C 180,E1 -19506.304,E2 -19506.304} C_VEL
LIN {X 0,Y 240.736,Z 495.513,A -85,B 0,C 180,E1 -19507.923,E2 -19507.923} C_VEL
LIN {X 0,Y 239.004,Z 505.064,A -85,B 0,C 180,E1 -19509.586,E2 -19509.586} C_VEL
LIN {X 0,Y 237.478,Z 514.468,A -85,B 0,C 180,E1 -19511.627,E2 -19511.627} C_VEL
LIN {X 0,Y 235.906,Z 523.273,A -85,B 0,C 180,E1 -19514.005,E2 -19514.005} C_VEL
LIN {X 0,Y 234.498,Z 530.846,A -85,B 0,C 180,E1 -19516.571,E2 -19516.571} C_VEL
LIN {X 0,Y 233.5,Z 537.841,A -85,B 0,C 180,E1 -19519.597,E2 -19519.597} C_VEL
LIN {X 0,Y 233.001,Z 542.44,A -85,B 0,C 180,E1 -19522.2,E2 -19522.2} C_VEL
LIN {X 0,Y 232.717,Z 546.41,A -85,B 0,C 180,E1 -19525.268,E2 -19525.268} C_VEL
LIN {X 0,Y 232.776,Z 548.971,A -85,B 0,C 180,E1 -19528.271,E2 -19528.271} C_VEL
LIN {X 0,Y 232.846,Z 549.886,A -85,B 0,C 180,E1 -19530.001,E2 -19530.001} C_VEL
LIN {X 0,Y 232.746,Z 550.394,A -85,B 0,C 180,E1 -19531.732,E2 -19531.732} C_VEL
LIN {X 0,Y 232.731,Z 550.162,A -85,B 0,C 180,E1 -19535.199,E2 -19535.199} C_VEL
LIN {X 0,Y 233.214,Z 548.4,A -85,B 0,C 180,E1 -19538.667,E2 -19538.667} C_VEL
LIN {X 0,Y 233.715,Z 546.887,A -85,B 0,C 180,E1 -19540.396,E2 -19540.396} C_VEL
LIN {X 0,Y 234.732,Z 543.848,A -85,B 0,C 180,E1 -19542.978,E2 -19542.978} C_VEL
LIN {X 0,Y 236.23,Z 539.779,A -85,B 0,C 180,E1 -19545.532,E2 -19545.532} C_VEL
LIN {X 0,Y 238.67,Z 533.561,A -85,B 0,C 180,E1 -19548.456,E2 -19548.456} C_VEL
LIN {X 0,Y 241.08,Z 526.777,A -85,B 0,C 180,E1 -19550.939,E2 -19550.939} C_VEL
LIN {X 0,Y 243.861,Z 518.474,A -85,B 0,C 180,E1 -19553.346,E2 -19553.346} C_VEL
LIN {X 0,Y 246.71,Z 509.893,A -85,B 0,C 180,E1 -19555.298,E2 -19555.298} C_VEL
LIN {X 0,Y 249.806,Z 499.351,A -85,B 0,C 180,E1 -19557.206,E2 -19557.206} C_VEL
LIN {X 0,Y 252.518,Z 488.909,A -85,B 0,C 180,E1 -19558.693,E2 -19558.693} C_VEL
LIN {X 0,Y 255.105,Z 477.388,A -85,B 0,C 180,E1 -19559.957,E2 -19559.957} C_VEL
LIN {X 0,Y 257.436,Z 464.163,A -85,B 0,C 180,E1 -19561.018,E2 -19561.018} C_VEL
LIN {X 0,Y 259.037,Z 451.717,A -85,B 0,C 180,E1 -19561.711,E2 -19561.711} C_VEL
LIN {X 0,Y 259.956,Z 438.456,A -85,B 0,C 180,E1 -19562.175,E2 -19562.175} C_VEL
LIN {X 0,Y 261.887,Z 392.533,A -85,B 0,C 180,E1 -19563.418,E2 -19563.418} C_VEL
LIN {X 0,Y 259.482,Z 378.574,A -85,B 0,C 180,E1 -19564.315,E2 -19564.315} C_VEL
LIN {X 0,Y 252.606,Z 363.351,A -85,B 0,C 180,E1 -19566.127,E2 -19566.127} C_VEL
LIN {X 0,Y 245.398,Z 349.69,A -85,B 0,C 180,E1 -19568.11,E2 -19568.11} C_VEL
LIN {X 0,Y 242.888,Z 345.343,A -85,B 0,C 180,E1 -19568.828,E2 -19568.828} C_VEL
LIN {X 0,Y 240.229,Z 340.796,A -85,B 0,C 180,E1 -19569.612,E2 -19569.612} C_VEL
LIN {X 0,Y 237.944,Z 336.723,A -85,B 0,C 180,E1 -19570.326,E2 -19570.326} C_VEL
LIN {X 0,Y 235.787,Z 329.379,A -85,B 0,C 180,E1 -19574.328,E2 -19574.328} C_VEL
LIN {X 0,Y 234.88,Z 326.223,A -85,B 0,C 180,E1 -19576.277,E2 -19576.277} C_VEL
LIN {X 0,Y 234.92,Z 326.217,A -85,B 0,C 180,E1 -19581.079,E2 -19581.079} C_VEL
LIN {X 0,Y 234.931,Z 326.215,A -85,B 0,C 180,E1 -19585.362,E2 -19585.362} C_VEL
LIN {X 0,Y 234.901,Z 326.225,A -85,B 0,C 180,E1 -19589.428,E2 -19589.428} C_VEL
LIN {X 0,Y 234.971,Z 326.215,A -85,B 0,C 180,E1 -19593.807,E2 -19593.807} C_VEL
LIN {X 0,Y 234.972,Z 326.207,A -85,B 0,C 180,E1 -19598.966,E2 -19598.966} C_VEL
LIN {X 0,Y 235.059,Z 326.194,A -85,B 0,C 180,E1 -19603.093,E2 -19603.093} C_VEL
LIN {X 0,Y 235.102,Z 326.187,A -85,B 0,C 180,E1 -19607.922,E2 -19607.922} C_VEL
LIN {X 0,Y 235.329,Z 326.157,A -85,B 0,C 180,E1 -19611.413,E2 -19611.413} C_VEL
LIN {X 0,Y 235.369,Z 326.158,A -85,B 0,C 180,E1 -19613.141,E2 -19613.141} C_VEL
LIN {X 0,Y 235.585,Z 326.135,A -85,B 0,C 180,E1 -19618.291,E2 -19618.291} C_VEL
LIN {X 0,Y 235.593,Z 326.129,A -85,B 0,C 180,E1 -19621.71,E2 -19621.71} C_VEL
LIN {X 0,Y 235.361,Z 326.166,A -85,B 0,C 180,E1 -19626.86,E2 -19626.86} C_VEL
LIN {X 0,Y 235.217,Z 326.178,A -85,B 0,C 180,E1 -19630.328,E2 -19630.328} C_VEL
LIN {X 0,Y 235.089,Z 326.201,A -85,B 0,C 180,E1 -19635.609,E2 -19635.609} C_VEL
LIN {X 0,Y 234.994,Z 326.212,A -85,B 0,C 180,E1 -19639.207,E2 -19639.207} C_VEL
LIN {X 0,Y 234.953,Z 326.214,A -85,B 0,C 180,E1 -19642.884,E2 -19642.884} C_VEL
LIN {X 0,Y 234.95,Z 326.215,A -85,B 0,C 180,E1 -19646.66,E2 -19646.66} C_VEL
LIN {X 0,Y 234.903,Z 326.222,A -85,B 0,C 180,E1 -19650.572,E2 -19650.572} C_VEL
LIN {X 0,Y 234.937,Z 326.214,A -85,B 0,C 180,E1 -19654.638,E2 -19654.638} C_VEL
LIN {X 0,Y 234.973,Z 326.306,A -85,B 0,C 180,E1 -19657.413,E2 -19657.413} C_VEL
LIN {X 0,Y 235.213,Z 327.449,A -85,B 0,C 180,E1 -19658.044,E2 -19658.044} C_VEL
LIN {X 0,Y 236.689,Z 330.034,A -85,B 0,C 180,E1 -19658.522,E2 -19658.522} C_VEL
LIN {X 0,Y 238.994,Z 333.324,A -85,B 0,C 180,E1 -19659.216,E2 -19659.216} C_VEL
LIN {X 0,Y 245.076,Z 343.019,A -85,B 0,C 180,E1 -19660.985,E2 -19660.985} C_VEL
LIN {X 0,Y 252.598,Z 356.145,A -85,B 0,C 180,E1 -19663.032,E2 -19663.032} C_VEL
LIN {X 0,Y 260.235,Z 371.691,A -85,B 0,C 180,E1 -19665.004,E2 -19665.004} C_VEL
LIN {X 0,Y 262.569,Z 377.06,A -85,B 0,C 180,E1 -19665.595,E2 -19665.595} C_VEL
LIN {X 0,Y 259.885,Z 434.744,A -85,B 0,C 180,E1 -19667.17,E2 -19667.17} C_VEL
LIN {X 0,Y 258.537,Z 447.594,A -85,B 0,C 180,E1 -19667.781,E2 -19667.781} C_VEL
LIN {X 0,Y 256.789,Z 459.985,A -85,B 0,C 180,E1 -19668.679,E2 -19668.679} C_VEL
LIN {X 0,Y 255,Z 469.812,A -85,B 0,C 180,E1 -19669.632,E2 -19669.632} C_VEL
LIN {X 0,Y 252.446,Z 481.711,A -85,B 0,C 180,E1 -19671.135,E2 -19671.135} C_VEL
LIN {X 0,Y 249.424,Z 492.98,A -85,B 0,C 180,E1 -19672.966,E2 -19672.966} C_VEL
LIN {X 0,Y 246.721,Z 501.797,A -85,B 0,C 180,E1 -19674.771,E2 -19674.771} C_VEL
LIN {X 0,Y 244.001,Z 509.87,A -85,B 0,C 180,E1 -19676.82,E2 -19676.82} C_VEL
LIN {X 0,Y 241.148,Z 517.682,A -85,B 0,C 180,E1 -19679.334,E2 -19679.334} C_VEL
LIN {X 0,Y 238.509,Z 524.408,A -85,B 0,C 180,E1 -19682.129,E2 -19682.129} C_VEL
LIN {X 0,Y 236.787,Z 528.802,A -85,B 0,C 180,E1 -19684.508,E2 -19684.508} C_VEL
LIN {X 0,Y 235.209,Z 532.516,A -85,B 0,C 180,E1 -19687.142,E2 -19687.142} C_VEL
LIN {X 0,Y 234.432,Z 534.416,A -85,B 0,C 180,E1 -19688.914,E2 -19688.914} C_VEL
LIN {X 0,Y 233.736,Z 535.825,A -85,B 0,C 180,E1 -19690.685,E2 -19690.685} C_VEL
LIN {X 0,Y 233.248,Z 536.813,A -85,B 0,C 180,E1 -19692.463,E2 -19692.463} C_VEL
LIN {X 0,Y 232.883,Z 537.505,A -85,B 0,C 180,E1 -19694.953,E2 -19694.953} C_VEL
LIN {X 0,Y 232.545,Z 537.308,A -85,B 0,C 180,E1 -19697.785,E2 -19697.785} C_VEL
LIN {X 0,Y 232.493,Z 536.652,A -85,B 0,C 180,E1 -19699.549,E2 -19699.549} C_VEL
LIN {X 0,Y 232.553,Z 535.605,A -85,B 0,C 180,E1 -19701.308,E2 -19701.308} C_VEL
LIN {X 0,Y 232.724,Z 534.12,A -85,B 0,C 180,E1 -19703.061,E2 -19703.061} C_VEL
LIN {X 0,Y 233.096,Z 531.093,A -85,B 0,C 180,E1 -19705.676,E2 -19705.676} C_VEL
LIN {X 0,Y 233.557,Z 527.026,A -85,B 0,C 180,E1 -19708.274,E2 -19708.274} C_VEL
LIN {X 0,Y 234.555,Z 520.778,A -85,B 0,C 180,E1 -19711.286,E2 -19711.286} C_VEL
LIN {X 0,Y 235.779,Z 513.984,A -85,B 0,C 180,E1 -19713.844,E2 -19713.844} C_VEL
LIN {X 0,Y 237.081,Z 507.055,A -85,B 0,C 180,E1 -19715.954,E2 -19715.954} C_VEL
LIN {X 0,Y 238.557,Z 498.725,A -85,B 0,C 180,E1 -19718.043,E2 -19718.043} C_VEL
LIN {X 0,Y 240.361,Z 489.586,A -85,B 0,C 180,E1 -19719.89,E2 -19719.89} C_VEL
LIN {X 0,Y 242.23,Z 478.242,A -85,B 0,C 180,E1 -19721.717,E2 -19721.717} C_VEL
LIN {X 0,Y 243.692,Z 467.164,A -85,B 0,C 180,E1 -19723.126,E2 -19723.126} C_VEL
LIN {X 0,Y 244.974,Z 454.851,A -85,B 0,C 180,E1 -19724.325,E2 -19724.325} C_VEL
LIN {X 0,Y 246.033,Z 441.713,A -85,B 0,C 180,E1 -19725.214,E2 -19725.214} C_VEL
LIN {X 0,Y 246.762,Z 428.986,A -85,B 0,C 180,E1 -19725.75,E2 -19725.75} C_VEL
LIN {X 0,Y 248.95,Z 363.935,A -85,B 0,C 180,E1 -19727.565,E2 -19727.565} C_VEL
LIN {X 0,Y 247.84,Z 358.786,A -85,B 0,C 180,E1 -19727.843,E2 -19727.843} C_VEL
LIN {X 0,Y 242.379,Z 343.84,A -85,B 0,C 180,E1 -19728.921,E2 -19728.921} C_VEL
LIN {X 0,Y 236.095,Z 329.248,A -85,B 0,C 180,E1 -19730.148,E2 -19730.148} C_VEL
LIN {X 0,Y 234.963,Z 326.343,A -85,B 0,C 180,E1 -19730.429,E2 -19730.429} C_VEL
LIN {X 0,Y 234.916,Z 326.224,A -85,B 0,C 180,E1 -19734.76,E2 -19734.76} C_VEL
LIN {X 0,Y 234.891,Z 326.226,A -85,B 0,C 180,E1 -19738.6,E2 -19738.6} C_VEL
LIN {X 0,Y 234.939,Z 326.217,A -85,B 0,C 180,E1 -19743.112,E2 -19743.112} C_VEL
LIN {X 0,Y 234.914,Z 326.222,A -85,B 0,C 180,E1 -19746.75,E2 -19746.75} C_VEL
LIN {X 0,Y 234.909,Z 326.222,A -85,B 0,C 180,E1 -19748.933,E2 -19748.933} C_VEL
LIN {X 0,Y 234.85,Z 326.23,A -85,B 0,C 180,E1 -19753.492,E2 -19753.492} C_VEL
LIN {X 0,Y 234.849,Z 326.223,A -85,B 0,C 180,E1 -19756.504,E2 -19756.504} C_VEL
LIN {X 0,Y 234.914,Z 326.223,A -85,B 0,C 180,E1 -19761.077,E2 -19761.077} C_VEL
LIN {X 0,Y 234.92,Z 326.209,A -85,B 0,C 180,E1 -19765.36,E2 -19765.36} C_VEL
LIN {X 0,Y 234.889,Z 326.226,A -85,B 0,C 180,E1 -19769.426,E2 -19769.426} C_VEL
LIN {X 0,Y 234.934,Z 326.203,A -85,B 0,C 180,E1 -19773.82,E2 -19773.82} C_VEL
LIN {X 0,Y 234.929,Z 326.219,A -85,B 0,C 180,E1 -19778.962,E2 -19778.962} C_VEL
LIN {X 0,Y 235.043,Z 326.197,A -85,B 0,C 180,E1 -19783.097,E2 -19783.097} C_VEL
LIN {X 0,Y 235.073,Z 326.199,A -85,B 0,C 180,E1 -19787.919,E2 -19787.919} C_VEL
LIN {X 0,Y 235.289,Z 326.174,A -85,B 0,C 180,E1 -19791.41,E2 -19791.41} C_VEL
LIN {X 0,Y 235.334,Z 326.162,A -85,B 0,C 180,E1 -19793.139,E2 -19793.139} C_VEL
LIN {X 0,Y 235.57,Z 326.136,A -85,B 0,C 180,E1 -19798.29,E2 -19798.29} C_VEL
LIN {X 0,Y 235.572,Z 326.139,A -85,B 0,C 180,E1 -19801.709,E2 -19801.709} C_VEL
LIN {X 0,Y 235.349,Z 326.156,A -85,B 0,C 180,E1 -19806.86,E2 -19806.86} C_VEL
LIN {X 0,Y 235.202,Z 326.186,A -85,B 0,C 180,E1 -19810.328,E2 -19810.328} C_VEL
LIN {X 0,Y 235.072,Z 326.187,A -85,B 0,C 180,E1 -19815.609,E2 -19815.609} C_VEL
LIN {X 0,Y 234.974,Z 326.215,A -85,B 0,C 180,E1 -19819.064,E2 -19819.064} C_VEL
LIN {X 0,Y 234.369,Z 326.302,A -85,B 0,C 180,E1 -19820.494,E2 -19820.494} C_VEL
LIN {X 0,Y 231.591,Z 326.654,A -85,B 0,C 180,E1 -19822.828,E2 -19822.828} C_VEL
LIN {X 0,Y 228.308,Z 327.05,A -85,B 0,C 180,E1 -19825.709,E2 -19825.709} C_VEL
LIN {X 0,Y 227.923,Z 327.092,A -85,B 0,C 180,E1 -19826.707,E2 -19826.707} C_VEL
LIN {X 0,Y 227.889,Z 327.095,A -85,B 0,C 180,E1 -19830.291,E2 -19830.291} C_VEL
LIN {X 0,Y 227.871,Z 327.098,A -85,B 0,C 180,E1 -19833.721,E2 -19833.721} C_VEL
LIN {X 0,Y 227.834,Z 327.104,A -85,B 0,C 180,E1 -19838.093,E2 -19838.093} C_VEL
LIN {X 0,Y 227.798,Z 327.1,A -85,B 0,C 180,E1 -19842.745,E2 -19842.745} C_VEL
LIN {X 0,Y 227.805,Z 327.108,A -85,B 0,C 180,E1 -19847.259,E2 -19847.259} C_VEL
LIN {X 0,Y 227.844,Z 327.104,A -85,B 0,C 180,E1 -19851.911,E2 -19851.911} C_VEL
LIN {X 0,Y 227.915,Z 327.144,A -85,B 0,C 180,E1 -19853.523,E2 -19853.523} C_VEL
LIN {X 0,Y 229.801,Z 335.561,A -85,B 0,C 180,E1 -19857.142,E2 -19857.142} C_VEL
LIN {X 0,Y 230.325,Z 338.015,A -85,B 0,C 180,E1 -19858.058,E2 -19858.058} C_VEL
LIN {X 0,Y 236.924,Z 355.103,A -85,B 0,C 180,E1 -19859.451,E2 -19859.451} C_VEL
LIN {X 0,Y 238.242,Z 359.464,A -85,B 0,C 180,E1 -19859.749,E2 -19859.749} C_VEL
LIN {X 0,Y 241.785,Z 388.845,A -85,B 0,C 180,E1 -19861.101,E2 -19861.101} C_VEL
LIN {X 0,Y 239.918,Z 446.847,A -85,B 0,C 180,E1 -19862.821,E2 -19862.821} C_VEL
LIN {X 0,Y 238.831,Z 460.711,A -85,B 0,C 180,E1 -19863.573,E2 -19863.573} C_VEL
LIN {X 0,Y 237.375,Z 473.119,A -85,B 0,C 180,E1 -19864.578,E2 -19864.578} C_VEL
LIN {X 0,Y 235.586,Z 485.83,A -85,B 0,C 180,E1 -19866.019,E2 -19866.019} C_VEL
LIN {X 0,Y 233.612,Z 497.124,A -85,B 0,C 180,E1 -19867.68,E2 -19867.68} C_VEL
LIN {X 0,Y 232,Z 506.271,A -85,B 0,C 180,E1 -19869.382,E2 -19869.382} C_VEL
LIN {X 0,Y 230.432,Z 515.409,A -85,B 0,C 180,E1 -19871.487,E2 -19871.487} C_VEL
LIN {X 0,Y 228.787,Z 524.031,A -85,B 0,C 180,E1 -19873.952,E2 -19873.952} C_VEL
LIN {X 0,Y 227.361,Z 531.436,A -85,B 0,C 180,E1 -19876.596,E2 -19876.596} C_VEL
LIN {X 0,Y 226.498,Z 537.373,A -85,B 0,C 180,E1 -19879.272,E2 -19879.272} C_VEL
LIN {X 0,Y 225.948,Z 542.035,A -85,B 0,C 180,E1 -19881.955,E2 -19881.955} C_VEL
LIN {X 0,Y 225.648,Z 545.565,A -85,B 0,C 180,E1 -19884.64,E2 -19884.64} C_VEL
LIN {X 0,Y 225.614,Z 547.345,A -85,B 0,C 180,E1 -19886.429,E2 -19886.429} C_VEL
LIN {X 0,Y 225.688,Z 548.687,A -85,B 0,C 180,E1 -19888.217,E2 -19888.217} C_VEL
LIN {X 0,Y 225.756,Z 549.627,A -85,B 0,C 180,E1 -19890.001,E2 -19890.001} C_VEL
LIN {X 0,Y 225.659,Z 550.168,A -85,B 0,C 180,E1 -19891.786,E2 -19891.786} C_VEL
LIN {X 0,Y 225.598,Z 550.186,A -85,B 0,C 180,E1 -19894.523,E2 -19894.523} C_VEL
LIN {X 0,Y 225.83,Z 549.334,A -85,B 0,C 180,E1 -19897.152,E2 -19897.152} C_VEL
LIN {X 0,Y 226.174,Z 548.288,A -85,B 0,C 180,E1 -19898.939,E2 -19898.939} C_VEL
LIN {X 0,Y 226.7,Z 546.823,A -85,B 0,C 180,E1 -19900.721,E2 -19900.721} C_VEL
LIN {X 0,Y 227.786,Z 543.833,A -85,B 0,C 180,E1 -19903.381,E2 -19903.381} C_VEL
LIN {X 0,Y 229.397,Z 539.816,A -85,B 0,C 180,E1 -19906.007,E2 -19906.007} C_VEL
LIN {X 0,Y 231.93,Z 533.666,A -85,B 0,C 180,E1 -19909.012,E2 -19909.012} C_VEL
LIN {X 0,Y 234.264,Z 527.456,A -85,B 0,C 180,E1 -19911.388,E2 -19911.388} C_VEL
LIN {X 0,Y 237.375,Z 518.742,A -85,B 0,C 180,E1 -19914.024,E2 -19914.024} C_VEL
LIN {X 0,Y 240.317,Z 510.289,A -85,B 0,C 180,E1 -19916.02,E2 -19916.02} C_VEL
LIN {X 0,Y 243.551,Z 499.874,A -85,B 0,C 180,E1 -19917.965,E2 -19917.965} C_VEL
LIN {X 0,Y 246.733,Z 488.172,A -85,B 0,C 180,E1 -19919.665,E2 -19919.665} C_VEL
LIN {X 0,Y 249.429,Z 476.445,A -85,B 0,C 180,E1 -19920.946,E2 -19920.946} C_VEL
LIN {X 0,Y 251.852,Z 462.993,A -85,B 0,C 180,E1 -19922.02,E2 -19922.02} C_VEL
LIN {X 0,Y 253.443,Z 450.162,A -85,B 0,C 180,E1 -19922.724,E2 -19922.724} C_VEL
LIN {X 0,Y 254.475,Z 434.021,A -85,B 0,C 180,E1 -19923.247,E2 -19923.247} C_VEL
LIN {X 0,Y 256.224,Z 393.513,A -85,B 0,C 180,E1 -19924.367,E2 -19924.367} C_VEL
LIN {X 0,Y 254.308,Z 381.718,A -85,B 0,C 180,E1 -19925.137,E2 -19925.137} C_VEL
LIN {X 0,Y 247.646,Z 366.991,A -85,B 0,C 180,E1 -19926.973,E2 -19926.973} C_VEL
LIN {X 0,Y 240.938,Z 354.026,A -85,B 0,C 180,E1 -19928.914,E2 -19928.914} C_VEL
LIN {X 0,Y 235.963,Z 345.398,A -85,B 0,C 180,E1 -19930.428,E2 -19930.428} C_VEL
LIN {X 0,Y 233.285,Z 341.003,A -85,B 0,C 180,E1 -19931.279,E2 -19931.279} C_VEL
LIN {X 0,Y 230.577,Z 336.317,A -85,B 0,C 180,E1 -19932.238,E2 -19932.238} C_VEL
LIN {X 0,Y 228.559,Z 329.508,A -85,B 0,C 180,E1 -19936.223,E2 -19936.223} C_VEL
LIN {X 0,Y 227.81,Z 327.107,A -85,B 0,C 180,E1 -19937.767,E2 -19937.767} C_VEL
LIN {X 0,Y 227.846,Z 327.096,A -85,B 0,C 180,E1 -19941.909,E2 -19941.909} C_VEL
LIN {X 0,Y 227.881,Z 327.099,A -85,B 0,C 180,E1 -19946.378,E2 -19946.378} C_VEL
LIN {X 0,Y 227.879,Z 327.096,A -85,B 0,C 180,E1 -19950.432,E2 -19950.432} C_VEL
LIN {X 0,Y 227.907,Z 327.091,A -85,B 0,C 180,E1 -19954.423,E2 -19954.423} C_VEL
LIN {X 0,Y 227.949,Z 327.085,A -85,B 0,C 180,E1 -19958.286,E2 -19958.286} C_VEL
LIN {X 0,Y 228.023,Z 327.071,A -85,B 0,C 180,E1 -19963.896,E2 -19963.896} C_VEL
LIN {X 0,Y 228.059,Z 327.063,A -85,B 0,C 180,E1 -19967.543,E2 -19967.543} C_VEL
LIN {X 0,Y 228.266,Z 327.038,A -85,B 0,C 180,E1 -19971.145,E2 -19971.145} C_VEL
LIN {X 0,Y 228.32,Z 327.035,A -85,B 0,C 180,E1 -19972.928,E2 -19972.928} C_VEL
LIN {X 0,Y 228.543,Z 327.013,A -85,B 0,C 180,E1 -19978.238,E2 -19978.238} C_VEL
LIN {X 0,Y 228.551,Z 327.006,A -85,B 0,C 180,E1 -19981.762,E2 -19981.762} C_VEL
LIN {X 0,Y 228.313,Z 327.043,A -85,B 0,C 180,E1 -19987.073,E2 -19987.073} C_VEL
LIN {X 0,Y 228.148,Z 327.062,A -85,B 0,C 180,E1 -19990.651,E2 -19990.651} C_VEL
LIN {X 0,Y 228.051,Z 327.069,A -85,B 0,C 180,E1 -19994.273,E2 -19994.273} C_VEL
LIN {X 0,Y 227.973,Z 327.077,A -85,B 0,C 180,E1 -19997.956,E2 -19997.956} C_VEL
LIN {X 0,Y 227.925,Z 327.085,A -85,B 0,C 180,E1 -20002.324,E2 -20002.324} C_VEL
LIN {X 0,Y 227.927,Z 327.09,A -85,B 0,C 180,E1 -20006.593,E2 -20006.593} C_VEL
LIN {X 0,Y 227.878,Z 327.098,A -85,B 0,C 180,E1 -20010.281,E2 -20010.281} C_VEL
LIN {X 0,Y 227.905,Z 327.09,A -85,B 0,C 180,E1 -20014.785,E2 -20014.785} C_VEL
LIN {X 0,Y 227.908,Z 327.227,A -85,B 0,C 180,E1 -20015.868,E2 -20015.868} C_VEL
LIN {X 0,Y 228.048,Z 327.918,A -85,B 0,C 180,E1 -20016.179,E2 -20016.179} C_VEL
LIN {X 0,Y 229.355,Z 330.609,A -85,B 0,C 180,E1 -20016.659,E2 -20016.659} C_VEL
LIN {X 0,Y 231.365,Z 332.798,A -85,B 0,C 180,E1 -20017.293,E2 -20017.293} C_VEL
LIN {X 0,Y 234.328,Z 337.179,A -85,B 0,C 180,E1 -20018.244,E2 -20018.244} C_VEL
LIN {X 0,Y 242.358,Z 350.24,A -85,B 0,C 180,E1 -20020.676,E2 -20020.676} C_VEL
LIN {X 0,Y 249.27,Z 363.017,A -85,B 0,C 180,E1 -20022.631,E2 -20022.631} C_VEL
LIN {X 0,Y 255.52,Z 376.076,A -85,B 0,C 180,E1 -20024.311,E2 -20024.311} C_VEL
LIN {X 0,Y 256.921,Z 379.346,A -85,B 0,C 180,E1 -20024.683,E2 -20024.683} C_VEL
LIN {X 0,Y 254.225,Z 434.674,A -85,B 0,C 180,E1 -20026.213,E2 -20026.213} C_VEL
LIN {X 0,Y 252.775,Z 448.047,A -85,B 0,C 180,E1 -20026.858,E2 -20026.858} C_VEL
LIN {X 0,Y 250.97,Z 460.375,A -85,B 0,C 180,E1 -20027.771,E2 -20027.771} C_VEL
LIN {X 0,Y 248.742,Z 471.893,A -85,B 0,C 180,E1 -20028.934,E2 -20028.934} C_VEL
LIN {X 0,Y 246.129,Z 483.19,A -85,B 0,C 180,E1 -20030.441,E2 -20030.441} C_VEL
LIN {X 0,Y 242.956,Z 494.355,A -85,B 0,C 180,E1 -20032.331,E2 -20032.331} C_VEL
LIN {X 0,Y 240.168,Z 502.954,A -85,B 0,C 180,E1 -20034.178,E2 -20034.178} C_VEL
LIN {X 0,Y 237.357,Z 510.827,A -85,B 0,C 180,E1 -20036.276,E2 -20036.276} C_VEL
LIN {X 0,Y 234.404,Z 518.488,A -85,B 0,C 180,E1 -20038.855,E2 -20038.855} C_VEL
LIN {X 0,Y 231.803,Z 524.741,A -85,B 0,C 180,E1 -20041.553,E2 -20041.553} C_VEL
LIN {X 0,Y 229.564,Z 530.07,A -85,B 0,C 180,E1 -20044.62,E2 -20044.62} C_VEL
LIN {X 0,Y 227.866,Z 533.872,A -85,B 0,C 180,E1 -20047.712,E2 -20047.712} C_VEL
LIN {X 0,Y 226.859,Z 535.893,A -85,B 0,C 180,E1 -20050.075,E2 -20050.075} C_VEL
LIN {X 0,Y 225.898,Z 537.546,A -85,B 0,C 180,E1 -20053.738,E2 -20053.738} C_VEL
LIN {X 0,Y 225.701,Z 537.774,A -85,B 0,C 180,E1 -20055.574,E2 -20055.574} C_VEL
LIN {X 0,Y 225.492,Z 537.567,A -85,B 0,C 180,E1 -20057.397,E2 -20057.397} C_VEL
LIN {X 0,Y 225.436,Z 535.939,A -85,B 0,C 180,E1 -20061.031,E2 -20061.031} C_VEL
LIN {X 0,Y 225.593,Z 534.526,A -85,B 0,C 180,E1 -20062.84,E2 -20062.84} C_VEL
LIN {X 0,Y 225.921,Z 531.975,A -85,B 0,C 180,E1 -20065.201,E2 -20065.201} C_VEL
LIN {X 0,Y 226.447,Z 527.585,A -85,B 0,C 180,E1 -20068.22,E2 -20068.22} C_VEL
LIN {X 0,Y 227.476,Z 521.446,A -85,B 0,C 180,E1 -20071.326,E2 -20071.326} C_VEL
LIN {X 0,Y 228.701,Z 514.758,A -85,B 0,C 180,E1 -20073.963,E2 -20073.963} C_VEL
LIN {X 0,Y 230.303,Z 506.463,A -85,B 0,C 180,E1 -20076.57,E2 -20076.57} C_VEL
LIN {X 0,Y 231.885,Z 497.938,A -85,B 0,C 180,E1 -20078.715,E2 -20078.715} C_VEL
LIN {X 0,Y 233.787,Z 488.547,A -85,B 0,C 180,E1 -20080.609,E2 -20080.609} C_VEL
LIN {X 0,Y 235.748,Z 476.927,A -85,B 0,C 180,E1 -20082.481,E2 -20082.481} C_VEL
LIN {X 0,Y 237.273,Z 465.463,A -85,B 0,C 180,E1 -20083.924,E2 -20083.924} C_VEL
LIN {X 0,Y 238.513,Z 453.597,A -85,B 0,C 180,E1 -20085.049,E2 -20085.049} C_VEL
LIN {X 0,Y 239.622,Z 439.858,A -85,B 0,C 180,E1 -20085.958,E2 -20085.958} C_VEL
LIN {X 0,Y 240.291,Z 427.209,A -85,B 0,C 180,E1 -20086.458,E2 -20086.458} C_VEL
LIN {X 0,Y 242.524,Z 364.991,A -85,B 0,C 180,E1 -20088.221,E2 -20088.221} C_VEL
LIN {X 0,Y 241.575,Z 360.96,A -85,B 0,C 180,E1 -20088.457,E2 -20088.457} C_VEL
LIN {X 0,Y 236.29,Z 346.467,A -85,B 0,C 180,E1 -20089.547,E2 -20089.547} C_VEL
LIN {X 0,Y 230.562,Z 333.047,A -85,B 0,C 180,E1 -20090.717,E2 -20090.717} C_VEL
LIN {X 0,Y 228.109,Z 328.093,A -85,B 0,C 180,E1 -20091.21,E2 -20091.21} C_VEL
LIN {X 0,Y 227.907,Z 327.099,A -85,B 0,C 180,E1 -20091.298,E2 -20091.298} C_VEL
LIN {X 0,Y 227.872,Z 327.1,A -85,B 0,C 180,E1 -20095.579,E2 -20095.579} C_VEL
LIN {X 0,Y 227.868,Z 327.099,A -85,B 0,C 180,E1 -20100.277,E2 -20100.277} C_VEL
LIN {X 0,Y 227.875,Z 327.097,A -85,B 0,C 180,E1 -20103.719,E2 -20103.719} C_VEL
LIN {X 0,Y 227.838,Z 327.104,A -85,B 0,C 180,E1 -20108.09,E2 -20108.09} C_VEL
LIN {X 0,Y 227.782,Z 327.11,A -85,B 0,C 180,E1 -20112.747,E2 -20112.747} C_VEL
LIN {X 0,Y 227.781,Z 327.1,A -85,B 0,C 180,E1 -20117.25,E2 -20117.25} C_VEL
LIN {X 0,Y 227.836,Z 327.1,A -85,B 0,C 180,E1 -20121.907,E2 -20121.907} C_VEL
LIN {X 0,Y 227.874,Z 327.089,A -85,B 0,C 180,E1 -20126.376,E2 -20126.376} C_VEL
LIN {X 0,Y 227.865,Z 327.097,A -85,B 0,C 180,E1 -20130.43,E2 -20130.43} C_VEL
LIN {X 0,Y 227.865,Z 327.082,A -85,B 0,C 180,E1 -20134.418,E2 -20134.418} C_VEL
LIN {X 0,Y 227.913,Z 327.094,A -85,B 0,C 180,E1 -20138.282,E2 -20138.282} C_VEL
LIN {X 0,Y 227.991,Z 327.067,A -85,B 0,C 180,E1 -20143.893,E2 -20143.893} C_VEL
LIN {X 0,Y 228.116,Z 327.067,A -85,B 0,C 180,E1 -20149.347,E2 -20149.347} C_VEL
LIN {X 0,Y 228.286,Z 327.039,A -85,B 0,C 180,E1 -20152.926,E2 -20152.926} C_VEL
LIN {X 0,Y 228.528,Z 327.012,A -85,B 0,C 180,E1 -20158.237,E2 -20158.237} C_VEL
LIN {X 0,Y 228.53,Z 327.016,A -85,B 0,C 180,E1 -20161.762,E2 -20161.762} C_VEL
LIN {X 0,Y 228.301,Z 327.035,A -85,B 0,C 180,E1 -20167.073,E2 -20167.073} C_VEL
LIN {X 0,Y 228.133,Z 327.069,A -85,B 0,C 180,E1 -20170.651,E2 -20170.651} C_VEL
LIN {X 0,Y 228.029,Z 327.071,A -85,B 0,C 180,E1 -20174.274,E2 -20174.274} C_VEL
LIN {X 0,Y 227.946,Z 327.085,A -85,B 0,C 180,E1 -20177.958,E2 -20177.958} C_VEL
LIN {X 0,Y 227.908,Z 327.092,A -85,B 0,C 180,E1 -20182.32,E2 -20182.32} C_VEL
LIN {X 0,Y 227.923,Z 327.092,A -85,B 0,C 180,E1 -20186.707,E2 -20186.707} C_VEL
LIN {X 0,Y 227.166,Z 327.182,A -85,B 0,C 180,E1 -20188.18,E2 -20188.18} C_VEL
LIN {X 0,Y 224.288,Z 327.544,A -85,B 0,C 180,E1 -20190.584,E2 -20190.584} C_VEL
LIN {X 0,Y 221.896,Z 327.842,A -85,B 0,C 180,E1 -20192.546,E2 -20192.546} C_VEL
LIN {X 0,Y 220.873,Z 327.97,A -85,B 0,C 180,E1 -20194.068,E2 -20194.068} C_VEL
LIN {X 0,Y 220.788,Z 327.98,A -85,B 0,C 180,E1 -20194.584,E2 -20194.584} C_VEL
LIN {X 0,Y 220.796,Z 327.978,A -85,B 0,C 180,E1 -20197.276,E2 -20197.276} C_VEL
LIN {X 0,Y 220.756,Z 327.975,A -85,B 0,C 180,E1 -20201.956,E2 -20201.956} C_VEL
LIN {X 0,Y 220.766,Z 327.986,A -85,B 0,C 180,E1 -20205.546,E2 -20205.546} C_VEL
LIN {X 0,Y 220.803,Z 327.981,A -85,B 0,C 180,E1 -20210.464,E2 -20210.464} C_VEL
LIN {X 0,Y 220.844,Z 328.098,A -85,B 0,C 180,E1 -20212.875,E2 -20212.875} C_VEL
LIN {X 0,Y 222.832,Z 336.747,A -85,B 0,C 180,E1 -20216.741,E2 -20216.741} C_VEL
LIN {X 0,Y 223.061,Z 337.739,A -85,B 0,C 180,E1 -20217.084,E2 -20217.084} C_VEL
LIN {X 0,Y 230.336,Z 356.17,A -85,B 0,C 180,E1 -20218.686,E2 -20218.686} C_VEL
LIN {X 0,Y 232.072,Z 361.878,A -85,B 0,C 180,E1 -20219.096,E2 -20219.096} C_VEL
LIN {X 0,Y 235.256,Z 388.557,A -85,B 0,C 180,E1 -20220.369,E2 -20220.369} C_VEL
LIN {X 0,Y 233.412,Z 446.15,A -85,B 0,C 180,E1 -20222.12,E2 -20222.12} C_VEL
LIN {X 0,Y 232.368,Z 459.414,A -85,B 0,C 180,E1 -20222.839,E2 -20222.839} C_VEL
LIN {X 0,Y 230.933,Z 471.579,A -85,B 0,C 180,E1 -20223.816,E2 -20223.816} C_VEL
LIN {X 0,Y 229.325,Z 483.058,A -85,B 0,C 180,E1 -20225.079,E2 -20225.079} C_VEL
LIN {X 0,Y 227.277,Z 494.834,A -85,B 0,C 180,E1 -20226.782,E2 -20226.782} C_VEL
LIN {X 0,Y 225.255,Z 505.41,A -85,B 0,C 180,E1 -20228.735,E2 -20228.735} C_VEL
LIN {X 0,Y 223.55,Z 515.136,A -85,B 0,C 180,E1 -20231.019,E2 -20231.019} C_VEL
LIN {X 0,Y 221.89,Z 523.414,A -85,B 0,C 180,E1 -20233.439,E2 -20233.439} C_VEL
LIN {X 0,Y 220.424,Z 530.896,A -85,B 0,C 180,E1 -20236.166,E2 -20236.166} C_VEL
LIN {X 0,Y 219.471,Z 536.896,A -85,B 0,C 180,E1 -20238.924,E2 -20238.924} C_VEL
LIN {X 0,Y 218.885,Z 541.619,A -85,B 0,C 180,E1 -20241.694,E2 -20241.694} C_VEL
LIN {X 0,Y 218.571,Z 545.205,A -85,B 0,C 180,E1 -20244.466,E2 -20244.466} C_VEL
LIN {X 0,Y 218.514,Z 547.035,A -85,B 0,C 180,E1 -20246.313,E2 -20246.313} C_VEL
LIN {X 0,Y 218.583,Z 548.402,A -85,B 0,C 180,E1 -20248.159,E2 -20248.159} C_VEL
LIN {X 0,Y 218.669,Z 549.368,A -85,B 0,C 180,E1 -20250.001,E2 -20250.001} C_VEL
LIN {X 0,Y 218.555,Z 549.933,A -85,B 0,C 180,E1 -20251.844,E2 -20251.844} C_VEL
LIN {X 0,Y 218.513,Z 550.025,A -85,B 0,C 180,E1 -20254.404,E2 -20254.404} C_VEL
LIN {X 0,Y 218.786,Z 549.196,A -85,B 0,C 180,E1 -20257.384,E2 -20257.384} C_VEL
LIN {X 0,Y 219.704,Z 546.754,A -85,B 0,C 180,E1 -20261.067,E2 -20261.067} C_VEL
LIN {X 0,Y 220.861,Z 543.806,A -85,B 0,C 180,E1 -20263.809,E2 -20263.809} C_VEL
LIN {X 0,Y 222.554,Z 539.841,A -85,B 0,C 180,E1 -20266.513,E2 -20266.513} C_VEL
LIN {X 0,Y 224.833,Z 534.764,A -85,B 0,C 180,E1 -20269.162,E2 -20269.162} C_VEL
LIN {X 0,Y 227.39,Z 528.404,A -85,B 0,C 180,E1 -20271.771,E2 -20271.771} C_VEL
LIN {X 0,Y 230.351,Z 520.486,A -85,B 0,C 180,E1 -20274.324,E2 -20274.324} C_VEL
LIN {X 0,Y 233.346,Z 512.436,A -85,B 0,C 180,E1 -20276.376,E2 -20276.376} C_VEL
LIN {X 0,Y 236.688,Z 502.635,A -85,B 0,C 180,E1 -20278.366,E2 -20278.366} C_VEL
LIN {X 0,Y 239.861,Z 491.695,A -85,B 0,C 180,E1 -20280.118,E2 -20280.118} C_VEL
LIN {X 0,Y 242.991,Z 479.231,A -85,B 0,C 180,E1 -20281.617,E2 -20281.617} C_VEL
LIN {X 0,Y 245.497,Z 466.961,A -85,B 0,C 180,E1 -20282.708,E2 -20282.708} C_VEL
LIN {X 0,Y 247.269,Z 454.865,A -85,B 0,C 180,E1 -20283.478,E2 -20283.478} C_VEL
LIN {X 0,Y 248.562,Z 441.363,A -85,B 0,C 180,E1 -20284.021,E2 -20284.021} C_VEL
LIN {X 0,Y 250.673,Z 394.856,A -85,B 0,C 180,E1 -20285.338,E2 -20285.338} C_VEL
LIN {X 0,Y 249.028,Z 384.562,A -85,B 0,C 180,E1 -20286.035,E2 -20286.035} C_VEL
LIN {X 0,Y 241.957,Z 368.849,A -85,B 0,C 180,E1 -20288.096,E2 -20288.096} C_VEL
LIN {X 0,Y 235.314,Z 356.105,A -85,B 0,C 180,E1 -20290.13,E2 -20290.13} C_VEL
LIN {X 0,Y 229.55,Z 346.303,A -85,B 0,C 180,E1 -20292.006,E2 -20292.006} C_VEL
LIN {X 0,Y 226.122,Z 340.858,A -85,B 0,C 180,E1 -20293.182,E2 -20293.182} C_VEL
LIN {X 0,Y 223.543,Z 336.73,A -85,B 0,C 180,E1 -20294.111,E2 -20294.111} C_VEL
LIN {X 0,Y 223.191,Z 335.928,A -85,B 0,C 180,E1 -20294.345,E2 -20294.345} C_VEL
LIN {X 0,Y 221.302,Z 329.931,A -85,B 0,C 180,E1 -20298.171,E2 -20298.171} C_VEL
LIN {X 0,Y 220.773,Z 327.981,A -85,B 0,C 180,E1 -20299.489,E2 -20299.489} C_VEL
LIN {X 0,Y 220.827,Z 327.976,A -85,B 0,C 180,E1 -20302.794,E2 -20302.794} C_VEL
LIN {X 0,Y 220.815,Z 327.973,A -85,B 0,C 180,E1 -20307.244,E2 -20307.244} C_VEL
LIN {X 0,Y 220.807,Z 327.972,A -85,B 0,C 180,E1 -20311.482,E2 -20311.482} C_VEL
LIN {X 0,Y 220.853,Z 327.966,A -85,B 0,C 180,E1 -20315.564,E2 -20315.564} C_VEL
LIN {X 0,Y 220.873,Z 327.962,A -85,B 0,C 180,E1 -20319.512,E2 -20319.512} C_VEL
LIN {X 0,Y 220.981,Z 327.947,A -85,B 0,C 180,E1 -20323.368,E2 -20323.368} C_VEL
LIN {X 0,Y 221.065,Z 327.942,A -85,B 0,C 180,E1 -20329.004,E2 -20329.004} C_VEL
LIN {X 0,Y 221.256,Z 327.912,A -85,B 0,C 180,E1 -20332.701,E2 -20332.701} C_VEL
LIN {X 0,Y 221.477,Z 327.893,A -85,B 0,C 180,E1 -20338.182,E2 -20338.182} C_VEL
LIN {X 0,Y 221.509,Z 327.884,A -85,B 0,C 180,E1 -20341.819,E2 -20341.819} C_VEL
LIN {X 0,Y 221.25,Z 327.923,A -85,B 0,C 180,E1 -20347.3,E2 -20347.3} C_VEL
LIN {X 0,Y 221.069,Z 327.947,A -85,B 0,C 180,E1 -20350.997,E2 -20350.997} C_VEL
LIN {X 0,Y 220.995,Z 327.95,A -85,B 0,C 180,E1 -20356.632,E2 -20356.632} C_VEL
LIN {X 0,Y 220.882,Z 327.964,A -85,B 0,C 180,E1 -20360.488,E2 -20360.488} C_VEL
LIN {X 0,Y 220.854,Z 327.965,A -85,B 0,C 180,E1 -20364.437,E2 -20364.437} C_VEL
LIN {X 0,Y 220.809,Z 327.969,A -85,B 0,C 180,E1 -20368.518,E2 -20368.518} C_VEL
LIN {X 0,Y 220.817,Z 327.975,A -85,B 0,C 180,E1 -20372.757,E2 -20372.757} C_VEL
LIN {X 0,Y 220.848,Z 327.97,A -85,B 0,C 180,E1 -20374.062,E2 -20374.062} C_VEL
LIN {X 0,Y 221.751,Z 330.656,A -85,B 0,C 180,E1 -20374.49,E2 -20374.49} C_VEL
LIN {X 0,Y 223.87,Z 332.952,A -85,B 0,C 180,E1 -20375.23,E2 -20375.23} C_VEL
LIN {X 0,Y 224.752,Z 334.349,A -85,B 0,C 180,E1 -20375.552,E2 -20375.552} C_VEL
LIN {X 0,Y 227.09,Z 337.472,A -85,B 0,C 180,E1 -20376.356,E2 -20376.356} C_VEL
LIN {X 0,Y 231.43,Z 343.971,A -85,B 0,C 180,E1 -20377.806,E2 -20377.806} C_VEL
LIN {X 0,Y 238.094,Z 354.914,A -85,B 0,C 180,E1 -20379.901,E2 -20379.901} C_VEL
LIN {X 0,Y 244.538,Z 366.973,A -85,B 0,C 180,E1 -20381.808,E2 -20381.808} C_VEL
LIN {X 0,Y 250.571,Z 379.738,A -85,B 0,C 180,E1 -20383.512,E2 -20383.512} C_VEL
LIN {X 0,Y 251.315,Z 381.371,A -85,B 0,C 180,E1 -20383.715,E2 -20383.715} C_VEL
LIN {X 0,Y 248.583,Z 435.234,A -85,B 0,C 180,E1 -20385.238,E2 -20385.238} C_VEL
LIN {X 0,Y 247.089,Z 448.503,A -85,B 0,C 180,E1 -20385.895,E2 -20385.895} C_VEL
LIN {X 0,Y 245.208,Z 460.761,A -85,B 0,C 180,E1 -20386.819,E2 -20386.819} C_VEL
LIN {X 0,Y 242.896,Z 472.225,A -85,B 0,C 180,E1 -20388.001,E2 -20388.001} C_VEL
LIN {X 0,Y 240.146,Z 483.577,A -85,B 0,C 180,E1 -20389.545,E2 -20389.545} C_VEL
LIN {X 0,Y 236.863,Z 494.639,A -85,B 0,C 180,E1 -20391.456,E2 -20391.456} C_VEL
LIN {X 0,Y 233.644,Z 504.056,A -85,B 0,C 180,E1 -20393.552,E2 -20393.552} C_VEL
LIN {X 0,Y 230.602,Z 512.087,A -85,B 0,C 180,E1 -20395.798,E2 -20395.798} C_VEL
LIN {X 0,Y 227.678,Z 519.303,A -85,B 0,C 180,E1 -20398.347,E2 -20398.347} C_VEL
LIN {X 0,Y 225.137,Z 525.066,A -85,B 0,C 180,E1 -20400.935,E2 -20400.935} C_VEL
LIN {X 0,Y 222.926,Z 529.968,A -85,B 0,C 180,E1 -20403.808,E2 -20403.808} C_VEL
LIN {X 0,Y 220.951,Z 534.144,A -85,B 0,C 180,E1 -20407.286,E2 -20407.286} C_VEL
LIN {X 0,Y 219.99,Z 535.948,A -85,B 0,C 180,E1 -20409.425,E2 -20409.425} C_VEL
LIN {X 0,Y 219.356,Z 537.027,A -85,B 0,C 180,E1 -20411.312,E2 -20411.312} C_VEL
LIN {X 0,Y 218.67,Z 537.958,A -85,B 0,C 180,E1 -20415.1,E2 -20415.1} C_VEL
LIN {X 0,Y 218.433,Z 537.823,A -85,B 0,C 180,E1 -20416.983,E2 -20416.983} C_VEL
LIN {X 0,Y 218.338,Z 536.273,A -85,B 0,C 180,E1 -20420.737,E2 -20420.737} C_VEL
LIN {X 0,Y 218.469,Z 534.904,A -85,B 0,C 180,E1 -20422.606,E2 -20422.606} C_VEL
LIN {X 0,Y 218.785,Z 532.753,A -85,B 0,C 180,E1 -20424.761,E2 -20424.761} C_VEL
LIN {X 0,Y 219.202,Z 529.544,A -85,B 0,C 180,E1 -20427.242,E2 -20427.242} C_VEL
LIN {X 0,Y 219.922,Z 524.893,A -85,B 0,C 180,E1 -20429.999,E2 -20429.999} C_VEL
LIN {X 0,Y 221.098,Z 517.894,A -85,B 0,C 180,E1 -20433.187,E2 -20433.187} C_VEL
LIN {X 0,Y 222.721,Z 510.302,A -85,B 0,C 180,E1 -20435.885,E2 -20435.885} C_VEL
LIN {X 0,Y 224.176,Z 502.561,A -85,B 0,C 180,E1 -20438.109,E2 -20438.109} C_VEL
LIN {X 0,Y 226.282,Z 492.014,A -85,B 0,C 180,E1 -20440.512,E2 -20440.512} C_VEL
LIN {X 0,Y 228.429,Z 481.241,A -85,B 0,C 180,E1 -20442.436,E2 -20442.436} C_VEL
LIN {X 0,Y 229.995,Z 470.827,A -85,B 0,C 180,E1 -20443.923,E2 -20443.923} C_VEL
LIN {X 0,Y 231.485,Z 458.339,A -85,B 0,C 180,E1 -20445.292,E2 -20445.292} C_VEL
LIN {X 0,Y 232.726,Z 445.144,A -85,B 0,C 180,E1 -20446.332,E2 -20446.332} C_VEL
LIN {X 0,Y 233.527,Z 433.075,A -85,B 0,C 180,E1 -20446.949,E2 -20446.949} C_VEL
LIN {X 0,Y 235.959,Z 364.952,A -85,B 0,C 180,E1 -20448.969,E2 -20448.969} C_VEL
LIN {X 0,Y 230.851,Z 350.63,A -85,B 0,C 180,E1 -20450.074,E2 -20450.074} C_VEL
LIN {X 0,Y 224.967,Z 336.727,A -85,B 0,C 180,E1 -20451.326,E2 -20451.326} C_VEL
LIN {X 0,Y 221.084,Z 329.086,A -85,B 0,C 180,E1 -20452.141,E2 -20452.141} C_VEL
LIN {X 0,Y 220.857,Z 327.973,A -85,B 0,C 180,E1 -20452.247,E2 -20452.247} C_VEL
LIN {X 0,Y 220.847,Z 327.975,A -85,B 0,C 180,E1 -20456.994,E2 -20456.994} C_VEL
LIN {X 0,Y 220.817,Z 327.977,A -85,B 0,C 180,E1 -20460.757,E2 -20460.757} C_VEL
LIN {X 0,Y 220.792,Z 327.981,A -85,B 0,C 180,E1 -20464.955,E2 -20464.955} C_VEL
LIN {X 0,Y 220.8,Z 327.981,A -85,B 0,C 180,E1 -20467.273,E2 -20467.273} C_VEL
LIN {X 0,Y 220.745,Z 327.982,A -85,B 0,C 180,E1 -20471.956,E2 -20471.956} C_VEL
LIN {X 0,Y 220.749,Z 327.981,A -85,B 0,C 180,E1 -20475.539,E2 -20475.539} C_VEL
LIN {X 0,Y 220.777,Z 327.981,A -85,B 0,C 180,E1 -20480.456,E2 -20480.456} C_VEL
LIN {X 0,Y 220.821,Z 327.973,A -85,B 0,C 180,E1 -20482.791,E2 -20482.791} C_VEL
LIN {X 0,Y 220.806,Z 327.973,A -85,B 0,C 180,E1 -20487.241,E2 -20487.241} C_VEL
LIN {X 0,Y 220.789,Z 327.975,A -85,B 0,C 180,E1 -20491.479,E2 -20491.479} C_VEL
LIN {X 0,Y 220.796,Z 327.967,A -85,B 0,C 180,E1 -20495.556,E2 -20495.556} C_VEL
LIN {X 0,Y 220.839,Z 327.977,A -85,B 0,C 180,E1 -20499.508,E2 -20499.508} C_VEL
LIN {X 0,Y 220.959,Z 327.946,A -85,B 0,C 180,E1 -20503.365,E2 -20503.365} C_VEL
LIN {X 0,Y 221.039,Z 327.948,A -85,B 0,C 180,E1 -20509.002,E2 -20509.002} C_VEL
LIN {X 0,Y 221.223,Z 327.919,A -85,B 0,C 180,E1 -20512.699,E2 -20512.699} C_VEL
LIN {X 0,Y 221.462,Z 327.892,A -85,B 0,C 180,E1 -20518.181,E2 -20518.181} C_VEL
LIN {X 0,Y 221.463,Z 327.897,A -85,B 0,C 180,E1 -20521.818,E2 -20521.818} C_VEL
LIN {X 0,Y 221.238,Z 327.916,A -85,B 0,C 180,E1 -20527.3,E2 -20527.3} C_VEL
LIN {X 0,Y 221.054,Z 327.949,A -85,B 0,C 180,E1 -20530.997,E2 -20530.997} C_VEL
LIN {X 0,Y 220.972,Z 327.944,A -85,B 0,C 180,E1 -20536.633,E2 -20536.633} C_VEL
LIN {X 0,Y 220.868,Z 327.972,A -85,B 0,C 180,E1 -20540.488,E2 -20540.488} C_VEL
LIN {X 0,Y 220.854,Z 327.97,A -85,B 0,C 180,E1 -20544.436,E2 -20544.436} C_VEL
LIN {X 0,Y 220.817,Z 327.972,A -85,B 0,C 180,E1 -20548.516,E2 -20548.516} C_VEL
LIN {X 0,Y 220.81,Z 327.976,A -85,B 0,C 180,E1 -20552.757,E2 -20552.757} C_VEL
LIN {X 0,Y 220.788,Z 327.98,A -85,B 0,C 180,E1 -20554.584,E2 -20554.584} C_VEL
LIN {X 0,Y 220.099,Z 328.068,A -85,B 0,C 180,E1 -20556.105,E2 -20556.105} C_VEL
LIN {X 0,Y 217.197,Z 328.429,A -85,B 0,C 180,E1 -20558.586,E2 -20558.586} C_VEL
LIN {X 0,Y 214.75,Z 328.73,A -85,B 0,C 180,E1 -20560.612,E2 -20560.612} C_VEL
LIN {X 0,Y 213.722,Z 328.85,A -85,B 0,C 180,E1 -20562.188,E2 -20562.188} C_VEL
LIN {X 0,Y 213.65,Z 328.859,A -85,B 0,C 180,E1 -20562.722,E2 -20562.722} C_VEL
LIN {X 0,Y 213.699,Z 328.865,A -85,B 0,C 180,E1 -20566.346,E2 -20566.346} C_VEL
LIN {X 0,Y 213.731,Z 328.863,A -85,B 0,C 180,E1 -20571.337,E2 -20571.337} C_VEL
LIN {X 0,Y 213.769,Z 328.865,A -85,B 0,C 180,E1 -20572.096,E2 -20572.096} C_VEL
LIN {X 0,Y 215.731,Z 337.215,A -85,B 0,C 180,E1 -20575.994,E2 -20575.994} C_VEL
LIN {X 0,Y 222.86,Z 354.864,A -85,B 0,C 180,E1 -20577.672,E2 -20577.672} C_VEL
LIN {X 0,Y 225.755,Z 363.142,A -85,B 0,C 180,E1 -20578.347,E2 -20578.347} C_VEL
LIN {X 0,Y 228.87,Z 390.053,A -85,B 0,C 180,E1 -20579.671,E2 -20579.671} C_VEL
LIN {X 0,Y 226.897,Z 446.527,A -85,B 0,C 180,E1 -20581.436,E2 -20581.436} C_VEL
LIN {X 0,Y 225.727,Z 460.366,A -85,B 0,C 180,E1 -20582.224,E2 -20582.224} C_VEL
LIN {X 0,Y 224.126,Z 473.269,A -85,B 0,C 180,E1 -20583.335,E2 -20583.335} C_VEL
LIN {X 0,Y 222.338,Z 485.069,A -85,B 0,C 180,E1 -20584.742,E2 -20584.742} C_VEL
LIN {X 0,Y 220.232,Z 496.434,A -85,B 0,C 180,E1 -20586.492,E2 -20586.492} C_VEL
LIN {X 0,Y 218.394,Z 505.623,A -85,B 0,C 180,E1 -20588.282,E2 -20588.282} C_VEL
LIN {X 0,Y 216.605,Z 515.344,A -85,B 0,C 180,E1 -20590.66,E2 -20590.66} C_VEL
LIN {X 0,Y 214.792,Z 524.168,A -85,B 0,C 180,E1 -20593.365,E2 -20593.365} C_VEL
LIN {X 0,Y 213.286,Z 531.481,A -85,B 0,C 180,E1 -20596.18,E2 -20596.18} C_VEL
LIN {X 0,Y 212.457,Z 536.417,A -85,B 0,C 180,E1 -20598.554,E2 -20598.554} C_VEL
LIN {X 0,Y 211.842,Z 541.202,A -85,B 0,C 180,E1 -20601.416,E2 -20601.416} C_VEL
LIN {X 0,Y 211.494,Z 544.844,A -85,B 0,C 180,E1 -20604.28,E2 -20604.28} C_VEL
LIN {X 0,Y 211.436,Z 546.717,A -85,B 0,C 180,E1 -20606.19,E2 -20606.19} C_VEL
LIN {X 0,Y 211.481,Z 548.118,A -85,B 0,C 180,E1 -20608.097,E2 -20608.097} C_VEL
LIN {X 0,Y 211.583,Z 549.109,A -85,B 0,C 180,E1 -20610.001,E2 -20610.001} C_VEL
LIN {X 0,Y 211.455,Z 549.697,A -85,B 0,C 180,E1 -20611.906,E2 -20611.906} C_VEL
LIN {X 0,Y 211.419,Z 549.868,A -85,B 0,C 180,E1 -20614.243,E2 -20614.243} C_VEL
LIN {X 0,Y 211.717,Z 549.058,A -85,B 0,C 180,E1 -20617.632,E2 -20617.632} C_VEL
LIN {X 0,Y 212.725,Z 546.677,A -85,B 0,C 180,E1 -20621.435,E2 -20621.435} C_VEL
LIN {X 0,Y 213.93,Z 543.773,A -85,B 0,C 180,E1 -20624.265,E2 -20624.265} C_VEL
LIN {X 0,Y 215.737,Z 539.864,A -85,B 0,C 180,E1 -20627.05,E2 -20627.05} C_VEL
LIN {X 0,Y 218.121,Z 534.848,A -85,B 0,C 180,E1 -20629.776,E2 -20629.776} C_VEL
LIN {X 0,Y 220.81,Z 528.575,A -85,B 0,C 180,E1 -20632.455,E2 -20632.455} C_VEL
LIN {X 0,Y 223.91,Z 520.75,A -85,B 0,C 180,E1 -20635.072,E2 -20635.072} C_VEL
LIN {X 0,Y 227.682,Z 511.019,A -85,B 0,C 180,E1 -20637.583,E2 -20637.583} C_VEL
LIN {X 0,Y 231.184,Z 500.935,A -85,B 0,C 180,E1 -20639.605,E2 -20639.605} C_VEL
LIN {X 0,Y 234.168,Z 490.966,A -85,B 0,C 180,E1 -20641.18,E2 -20641.18} C_VEL
LIN {X 0,Y 237.432,Z 478.374,A -85,B 0,C 180,E1 -20642.698,E2 -20642.698} C_VEL
LIN {X 0,Y 240.043,Z 465.816,A -85,B 0,C 180,E1 -20643.8,E2 -20643.8} C_VEL
LIN {X 0,Y 241.825,Z 454.005,A -85,B 0,C 180,E1 -20644.538,E2 -20644.538} C_VEL
LIN {X 0,Y 243.046,Z 440.768,A -85,B 0,C 180,E1 -20645.079,E2 -20645.079} C_VEL
LIN {X 0,Y 245.208,Z 395.865,A -85,B 0,C 180,E1 -20646.366,E2 -20646.366} C_VEL
LIN {X 0,Y 243.794,Z 387.407,A -85,B 0,C 180,E1 -20646.979,E2 -20646.979} C_VEL
LIN {X 0,Y 237.295,Z 372.814,A -85,B 0,C 180,E1 -20648.973,E2 -20648.973} C_VEL
LIN {X 0,Y 231.008,Z 360.547,A -85,B 0,C 180,E1 -20650.999,E2 -20650.999} C_VEL
LIN {X 0,Y 225.089,Z 350.458,A -85,B 0,C 180,E1 -20653.023,E2 -20653.023} C_VEL
LIN {X 0,Y 222.31,Z 345.89,A -85,B 0,C 180,E1 -20654.03,E2 -20654.03} C_VEL
LIN {X 0,Y 219.035,Z 340.812,A -85,B 0,C 180,E1 -20655.264,E2 -20655.264} C_VEL
LIN {X 0,Y 216.214,Z 336.569,A -85,B 0,C 180,E1 -20656.381,E2 -20656.381} C_VEL
LIN {X 0,Y 215.833,Z 335.677,A -85,B 0,C 180,E1 -20656.613,E2 -20656.613} C_VEL
LIN {X 0,Y 213.74,Z 328.853,A -85,B 0,C 180,E1 -20661.454,E2 -20661.454} C_VEL
LIN {X 0,Y 213.759,Z 328.857,A -85,B 0,C 180,E1 -20666.018,E2 -20666.018} C_VEL
LIN {X 0,Y 213.753,Z 328.855,A -85,B 0,C 180,E1 -20670.45,E2 -20670.45} C_VEL
LIN {X 0,Y 213.786,Z 328.847,A -85,B 0,C 180,E1 -20674.7,E2 -20674.7} C_VEL
LIN {X 0,Y 213.798,Z 328.844,A -85,B 0,C 180,E1 -20678.802,E2 -20678.802} C_VEL
LIN {X 0,Y 213.894,Z 328.83,A -85,B 0,C 180,E1 -20682.8,E2 -20682.8} C_VEL
LIN {X 0,Y 213.937,Z 328.824,A -85,B 0,C 180,E1 -20686.706,E2 -20686.706} C_VEL
LIN {X 0,Y 214.142,Z 328.801,A -85,B 0,C 180,E1 -20690.556,E2 -20690.556} C_VEL
LIN {X 0,Y 214.091,Z 328.81,A -85,B 0,C 180,E1 -20694.349,E2 -20694.349} C_VEL
LIN {X 0,Y 214.413,Z 328.772,A -85,B 0,C 180,E1 -20698.122,E2 -20698.122} C_VEL
LIN {X 0,Y 214.54,Z 328.746,A -85,B 0,C 180,E1 -20700,E2 -20700} C_VEL
LIN {X 0,Y 214.442,Z 328.764,A -85,B 0,C 180,E1 -20701.878,E2 -20701.878} C_VEL
LIN {X 0,Y 214.191,Z 328.802,A -85,B 0,C 180,E1 -20707.542,E2 -20707.542} C_VEL
LIN {X 0,Y 214.001,Z 328.828,A -85,B 0,C 180,E1 -20711.365,E2 -20711.365} C_VEL
LIN {X 0,Y 213.917,Z 328.839,A -85,B 0,C 180,E1 -20715.239,E2 -20715.239} C_VEL
LIN {X 0,Y 213.824,Z 328.848,A -85,B 0,C 180,E1 -20719.189,E2 -20719.189} C_VEL
LIN {X 0,Y 213.807,Z 328.851,A -85,B 0,C 180,E1 -20723.232,E2 -20723.232} C_VEL
LIN {X 0,Y 213.792,Z 328.848,A -85,B 0,C 180,E1 -20727.428,E2 -20727.428} C_VEL
LIN {X 0,Y 213.754,Z 328.903,A -85,B 0,C 180,E1 -20731.81,E2 -20731.81} C_VEL
LIN {X 0,Y 214.691,Z 331.603,A -85,B 0,C 180,E1 -20732.276,E2 -20732.276} C_VEL
LIN {X 0,Y 216.931,Z 333.919,A -85,B 0,C 180,E1 -20733.142,E2 -20733.142} C_VEL
LIN {X 0,Y 217.638,Z 334.794,A -85,B 0,C 180,E1 -20733.415,E2 -20733.415} C_VEL
LIN {X 0,Y 219.779,Z 337.986,A -85,B 0,C 180,E1 -20734.251,E2 -20734.251} C_VEL
LIN {X 0,Y 221.092,Z 339.497,A -85,B 0,C 180,E1 -20734.725,E2 -20734.725} C_VEL
LIN {X 0,Y 223.717,Z 343.143,A -85,B 0,C 180,E1 -20735.672,E2 -20735.672} C_VEL
LIN {X 0,Y 227.981,Z 349.729,A -85,B 0,C 180,E1 -20737.159,E2 -20737.159} C_VEL
LIN {X 0,Y 233.936,Z 359.701,A -85,B 0,C 180,E1 -20739.116,E2 -20739.116} C_VEL
LIN {X 0,Y 241.116,Z 373.415,A -85,B 0,C 180,E1 -20741.329,E2 -20741.329} C_VEL
LIN {X 0,Y 245.839,Z 383.835,A -85,B 0,C 180,E1 -20742.729,E2 -20742.729} C_VEL
LIN {X 0,Y 243.127,Z 434.753,A -85,B 0,C 180,E1 -20744.176,E2 -20744.176} C_VEL
LIN {X 0,Y 241.607,Z 448.229,A -85,B 0,C 180,E1 -20744.845,E2 -20744.845} C_VEL
LIN {X 0,Y 239.521,Z 461.15,A -85,B 0,C 180,E1 -20745.822,E2 -20745.822} C_VEL
LIN {X 0,Y 237.113,Z 472.556,A -85,B 0,C 180,E1 -20747.021,E2 -20747.021} C_VEL
LIN {X 0,Y 234.115,Z 484.369,A -85,B 0,C 180,E1 -20748.666,E2 -20748.666} C_VEL
LIN {X 0,Y 230.846,Z 494.924,A -85,B 0,C 180,E1 -20750.54,E2 -20750.54} C_VEL
LIN {X 0,Y 227.8,Z 503.488,A -85,B 0,C 180,E1 -20752.458,E2 -20752.458} C_VEL
LIN {X 0,Y 224.438,Z 511.995,A -85,B 0,C 180,E1 -20754.858,E2 -20754.858} C_VEL
LIN {X 0,Y 221.421,Z 518.975,A -85,B 0,C 180,E1 -20757.343,E2 -20757.343} C_VEL
LIN {X 0,Y 218.504,Z 525.386,A -85,B 0,C 180,E1 -20760.278,E2 -20760.278} C_VEL
LIN {X 0,Y 216.343,Z 529.839,A -85,B 0,C 180,E1 -20762.947,E2 -20762.947} C_VEL
LIN {X 0,Y 214.551,Z 533.443,A -85,B 0,C 180,E1 -20765.828,E2 -20765.828} C_VEL
LIN {X 0,Y 213.161,Z 535.981,A -85,B 0,C 180,E1 -20768.734,E2 -20768.734} C_VEL
LIN {X 0,Y 212.429,Z 537.136,A -85,B 0,C 180,E1 -20770.679,E2 -20770.679} C_VEL
LIN {X 0,Y 211.632,Z 538.142,A -85,B 0,C 180,E1 -20774.592,E2 -20774.592} C_VEL
LIN {X 0,Y 211.369,Z 538.057,A -85,B 0,C 180,E1 -20776.54,E2 -20776.54} C_VEL
LIN {X 0,Y 211.206,Z 537.542,A -85,B 0,C 180,E1 -20778.482,E2 -20778.482} C_VEL
LIN {X 0,Y 211.215,Z 536.606,A -85,B 0,C 180,E1 -20780.422,E2 -20780.422} C_VEL
LIN {X 0,Y 211.353,Z 535.274,A -85,B 0,C 180,E1 -20782.355,E2 -20782.355} C_VEL
LIN {X 0,Y 211.695,Z 532.896,A -85,B 0,C 180,E1 -20784.856,E2 -20784.856} C_VEL
LIN {X 0,Y 212.241,Z 528.646,A -85,B 0,C 180,E1 -20788.101,E2 -20788.101} C_VEL
LIN {X 0,Y 213.094,Z 523.7,A -85,B 0,C 180,E1 -20790.943,E2 -20790.943} C_VEL
LIN {X 0,Y 214.251,Z 517.489,A -85,B 0,C 180,E1 -20793.76,E2 -20793.76} C_VEL
LIN {X 0,Y 215.973,Z 509.716,A -85,B 0,C 180,E1 -20796.538,E2 -20796.538} C_VEL
LIN {X 0,Y 217.891,Z 500.022,A -85,B 0,C 180,E1 -20799.279,E2 -20799.279} C_VEL
LIN {X 0,Y 219.794,Z 491.046,A -85,B 0,C 180,E1 -20801.293,E2 -20801.293} C_VEL
LIN {X 0,Y 221.753,Z 481.33,A -85,B 0,C 180,E1 -20803.049,E2 -20803.049} C_VEL
LIN {X 0,Y 223.397,Z 470.88,A -85,B 0,C 180,E1 -20804.575,E2 -20804.575} C_VEL
LIN {X 0,Y 224.954,Z 458.344,A -85,B 0,C 180,E1 -20805.98,E2 -20805.98} C_VEL
LIN {X 0,Y 226.243,Z 445.079,A -85,B 0,C 180,E1 -20807.046,E2 -20807.046} C_VEL
LIN {X 0,Y 227.079,Z 432.769,A -85,B 0,C 180,E1 -20807.678,E2 -20807.678} C_VEL
LIN {X 0,Y 229.627,Z 366.711,A -85,B 0,C 180,E1 -20809.672,E2 -20809.672} C_VEL
LIN {X 0,Y 224.628,Z 352.822,A -85,B 0,C 180,E1 -20810.799,E2 -20810.799} C_VEL
LIN {X 0,Y 219.347,Z 340.294,A -85,B 0,C 180,E1 -20811.978,E2 -20811.978} C_VEL
LIN {X 0,Y 214.763,Z 331.656,A -85,B 0,C 180,E1 -20812.974,E2 -20812.974} C_VEL
LIN {X 0,Y 213.785,Z 328.855,A -85,B 0,C 180,E1 -20813.232,E2 -20813.232} C_VEL
LIN {X 0,Y 213.784,Z 328.854,A -85,B 0,C 180,E1 -20817.425,E2 -20817.425} C_VEL
LIN {X 0,Y 213.757,Z 328.857,A -85,B 0,C 180,E1 -20821.737,E2 -20821.737} C_VEL
LIN {X 0,Y 213.739,Z 328.858,A -85,B 0,C 180,E1 -20826.287,E2 -20826.287} C_VEL
LIN {X 0,Y 213.695,Z 328.858,A -85,B 0,C 180,E1 -20831.127,E2 -20831.127} C_VEL
LIN {X 0,Y 213.698,Z 328.864,A -85,B 0,C 180,E1 -20833.678,E2 -20833.678} C_VEL
LIN {X 0,Y 213.697,Z 328.856,A -85,B 0,C 180,E1 -20836.344,E2 -20836.344} C_VEL
LIN {X 0,Y 213.7,Z 328.863,A -85,B 0,C 180,E1 -20841.328,E2 -20841.328} C_VEL
LIN {X 0,Y 213.749,Z 328.846,A -85,B 0,C 180,E1 -20846.016,E2 -20846.016} C_VEL
LIN {X 0,Y 213.741,Z 328.856,A -85,B 0,C 180,E1 -20850.447,E2 -20850.447} C_VEL
LIN {X 0,Y 213.744,Z 328.84,A -85,B 0,C 180,E1 -20854.694,E2 -20854.694} C_VEL
LIN {X 0,Y 213.768,Z 328.855,A -85,B 0,C 180,E1 -20858.798,E2 -20858.798} C_VEL
LIN {X 0,Y 213.871,Z 328.833,A -85,B 0,C 180,E1 -20862.797,E2 -20862.797} C_VEL
LIN {X 0,Y 213.894,Z 328.832,A -85,B 0,C 180,E1 -20866.702,E2 -20866.702} C_VEL
LIN {X 0,Y 214.116,Z 328.812,A -85,B 0,C 180,E1 -20870.554,E2 -20870.554} C_VEL
LIN {X 0,Y 214.066,Z 328.799,A -85,B 0,C 180,E1 -20874.347,E2 -20874.347} C_VEL
LIN {X 0,Y 214.398,Z 328.771,A -85,B 0,C 180,E1 -20878.121,E2 -20878.121} C_VEL
LIN {X 0,Y 214.504,Z 328.764,A -85,B 0,C 180,E1 -20880,E2 -20880} C_VEL
LIN {X 0,Y 214.4,Z 328.777,A -85,B 0,C 180,E1 -20881.878,E2 -20881.878} C_VEL
LIN {X 0,Y 214.179,Z 328.795,A -85,B 0,C 180,E1 -20887.542,E2 -20887.542} C_VEL
LIN {X 0,Y 213.985,Z 328.828,A -85,B 0,C 180,E1 -20891.365,E2 -20891.365} C_VEL
LIN {X 0,Y 213.894,Z 328.823,A -85,B 0,C 180,E1 -20895.24,E2 -20895.24} C_VEL
LIN {X 0,Y 213.807,Z 328.853,A -85,B 0,C 180,E1 -20899.19,E2 -20899.19} C_VEL
LIN {X 0,Y 213.804,Z 328.847,A -85,B 0,C 180,E1 -20903.232,E2 -20903.232} C_VEL
LIN {X 0,Y 213.823,Z 328.845,A -85,B 0,C 180,E1 -20907.45,E2 -20907.45} C_VEL
LIN {X 0,Y 213.761,Z 328.855,A -85,B 0,C 180,E1 -20911.738,E2 -20911.738} C_VEL
LIN {X 0,Y 213.735,Z 328.858,A -85,B 0,C 180,E1 -20916.29,E2 -20916.29} C_VEL
LIN {X 0,Y 213.699,Z 328.857,A -85,B 0,C 180,E1 -20921.128,E2 -20921.128} C_VEL
LIN {X 0,Y 213.65,Z 328.859,A -85,B 0,C 180,E1 -20922.722,E2 -20922.722} C_VEL
LIN {X 0,Y 213.003,Z 328.953,A -85,B 0,C 180,E1 -20924.296,E2 -20924.296} C_VEL
LIN {X 0,Y 210.143,Z 329.308,A -85,B 0,C 180,E1 -20926.866,E2 -20926.866} C_VEL
LIN {X 0,Y 207.731,Z 329.609,A -85,B 0,C 180,E1 -20928.967,E2 -20928.967} C_VEL
LIN {X 0,Y 206.747,Z 329.732,A -85,B 0,C 180,E1 -20930.6,E2 -20930.6} C_VEL
LIN {X 0,Y 206.696,Z 329.739,A -85,B 0,C 180,E1 -20931.152,E2 -20931.152} C_VEL
LIN {X 0,Y 206.739,Z 329.993,A -85,B 0,C 180,E1 -20931.432,E2 -20931.432} C_VEL
LIN {X 0,Y 208.437,Z 337.036,A -85,B 0,C 180,E1 -20934.877,E2 -20934.877} C_VEL
LIN {X 0,Y 216.466,Z 356.319,A -85,B 0,C 180,E1 -20936.837,E2 -20936.837} C_VEL
LIN {X 0,Y 219.735,Z 366.066,A -85,B 0,C 180,E1 -20937.653,E2 -20937.653} C_VEL
LIN {X 0,Y 222.489,Z 391.259,A -85,B 0,C 180,E1 -20938.922,E2 -20938.922} C_VEL
LIN {X 0,Y 220.434,Z 446.212,A -85,B 0,C 180,E1 -20940.676,E2 -20940.676} C_VEL
LIN {X 0,Y 219.269,Z 459.778,A -85,B 0,C 180,E1 -20941.462,E2 -20941.462} C_VEL
LIN {X 0,Y 217.608,Z 472.816,A -85,B 0,C 180,E1 -20942.6,E2 -20942.6} C_VEL
LIN {X 0,Y 215.615,Z 485.467,A -85,B 0,C 180,E1 -20944.155,E2 -20944.155} C_VEL
LIN {X 0,Y 213.435,Z 496.721,A -85,B 0,C 180,E1 -20945.955,E2 -20945.955} C_VEL
LIN {X 0,Y 211.397,Z 506.839,A -85,B 0,C 180,E1 -20948.039,E2 -20948.039} C_VEL
LIN {X 0,Y 209.58,Z 516.001,A -85,B 0,C 180,E1 -20950.409,E2 -20950.409} C_VEL
LIN {X 0,Y 207.671,Z 524.912,A -85,B 0,C 180,E1 -20953.284,E2 -20953.284} C_VEL
LIN {X 0,Y 206.12,Z 532.016,A -85,B 0,C 180,E1 -20956.193,E2 -20956.193} C_VEL
LIN {X 0,Y 205.187,Z 537.689,A -85,B 0,C 180,E1 -20959.143,E2 -20959.143} C_VEL
LIN {X 0,Y 204.637,Z 542.138,A -85,B 0,C 180,E1 -20962.106,E2 -20962.106} C_VEL
LIN {X 0,Y 204.351,Z 546.182,A -85,B 0,C 180,E1 -20965.836,E2 -20965.836} C_VEL
LIN {X 0,Y 204.382,Z 547.831,A -85,B 0,C 180,E1 -20968.031,E2 -20968.031} C_VEL
LIN {X 0,Y 204.498,Z 548.848,A -85,B 0,C 180,E1 -20970.001,E2 -20970.001} C_VEL
LIN {X 0,Y 204.357,Z 549.461,A -85,B 0,C 180,E1 -20971.972,E2 -20971.972} C_VEL
LIN {X 0,Y 204.321,Z 549.696,A -85,B 0,C 180,E1 -20974.046,E2 -20974.046} C_VEL
LIN {X 0,Y 204.666,Z 548.921,A -85,B 0,C 180,E1 -20977.896,E2 -20977.896} C_VEL
LIN {X 0,Y 205.747,Z 546.591,A -85,B 0,C 180,E1 -20981.828,E2 -20981.828} C_VEL
LIN {X 0,Y 207.025,Z 543.74,A -85,B 0,C 180,E1 -20984.752,E2 -20984.752} C_VEL
LIN {X 0,Y 208.947,Z 539.888,A -85,B 0,C 180,E1 -20987.622,E2 -20987.622} C_VEL
LIN {X 0,Y 211.419,Z 534.932,A -85,B 0,C 180,E1 -20990.43,E2 -20990.43} C_VEL
LIN {X 0,Y 214.55,Z 527.976,A -85,B 0,C 180,E1 -20993.481,E2 -20993.481} C_VEL
LIN {X 0,Y 218.127,Z 519.536,A -85,B 0,C 180,E1 -20996.298,E2 -20996.298} C_VEL
LIN {X 0,Y 221.444,Z 511.379,A -85,B 0,C 180,E1 -20998.429,E2 -20998.429} C_VEL
LIN {X 0,Y 225.078,Z 501.45,A -85,B 0,C 180,E1 -21000.492,E2 -21000.492} C_VEL
LIN {X 0,Y 228.583,Z 490.252,A -85,B 0,C 180,E1 -21002.291,E2 -21002.291} C_VEL
LIN {X 0,Y 231.522,Z 479.302,A -85,B 0,C 180,E1 -21003.642,E2 -21003.642} C_VEL
LIN {X 0,Y 234.201,Z 467.18,A -85,B 0,C 180,E1 -21004.762,E2 -21004.762} C_VEL
LIN {X 0,Y 236.221,Z 454.734,A -85,B 0,C 180,E1 -21005.581,E2 -21005.581} C_VEL
LIN {X 0,Y 237.573,Z 441.4,A -85,B 0,C 180,E1 -21006.143,E2 -21006.143} C_VEL
LIN {X 0,Y 239.818,Z 397.065,A -85,B 0,C 180,E1 -21007.437,E2 -21007.437} C_VEL
LIN {X 0,Y 238.838,Z 390.785,A -85,B 0,C 180,E1 -21007.899,E2 -21007.899} C_VEL
LIN {X 0,Y 232.653,Z 376.671,A -85,B 0,C 180,E1 -21009.898,E2 -21009.898} C_VEL
LIN {X 0,Y 226.577,Z 364.711,A -85,B 0,C 180,E1 -21011.962,E2 -21011.962} C_VEL
LIN {X 0,Y 221.373,Z 355.615,A -85,B 0,C 180,E1 -21013.835,E2 -21013.835} C_VEL
LIN {X 0,Y 218.449,Z 350.799,A -85,B 0,C 180,E1 -21014.945,E2 -21014.945} C_VEL
LIN {X 0,Y 215.393,Z 346.001,A -85,B 0,C 180,E1 -21016.158,E2 -21016.158} C_VEL
LIN {X 0,Y 211.86,Z 340.63,A -85,B 0,C 180,E1 -21017.637,E2 -21017.637} C_VEL
LIN {X 0,Y 208.755,Z 336.177,A -85,B 0,C 180,E1 -21019.01,E2 -21019.01} C_VEL
LIN {X 0,Y 208.404,Z 335.385,A -85,B 0,C 180,E1 -21019.22,E2 -21019.22} C_VEL
LIN {X 0,Y 206.701,Z 329.734,A -85,B 0,C 180,E1 -21023.638,E2 -21023.638} C_VEL
LIN {X 0,Y 206.712,Z 329.727,A -85,B 0,C 180,E1 -21028.211,E2 -21028.211} C_VEL
LIN {X 0,Y 206.712,Z 329.728,A -85,B 0,C 180,E1 -21032.127,E2 -21032.127} C_VEL
LIN {X 0,Y 206.749,Z 329.729,A -85,B 0,C 180,E1 -21036.61,E2 -21036.61} C_VEL
LIN {X 0,Y 206.827,Z 329.714,A -85,B 0,C 180,E1 -21042.193,E2 -21042.193} C_VEL
LIN {X 0,Y 206.878,Z 329.707,A -85,B 0,C 180,E1 -21046.243,E2 -21046.243} C_VEL
LIN {X 0,Y 207.103,Z 329.68,A -85,B 0,C 180,E1 -21050.231,E2 -21050.231} C_VEL
LIN {X 0,Y 207.054,Z 329.687,A -85,B 0,C 180,E1 -21054.156,E2 -21054.156} C_VEL
LIN {X 0,Y 207.353,Z 329.65,A -85,B 0,C 180,E1 -21058.058,E2 -21058.058} C_VEL
LIN {X 0,Y 207.505,Z 329.621,A -85,B 0,C 180,E1 -21060,E2 -21060} C_VEL
LIN {X 0,Y 207.378,Z 329.644,A -85,B 0,C 180,E1 -21061.943,E2 -21061.943} C_VEL
LIN {X 0,Y 207.135,Z 329.678,A -85,B 0,C 180,E1 -21067.801,E2 -21067.801} C_VEL
LIN {X 0,Y 206.925,Z 329.709,A -85,B 0,C 180,E1 -21071.759,E2 -21071.759} C_VEL
LIN {X 0,Y 206.85,Z 329.719,A -85,B 0,C 180,E1 -21075.773,E2 -21075.773} C_VEL
LIN {X 0,Y 206.861,Z 329.706,A -85,B 0,C 180,E1 -21077.955,E2 -21077.955} C_VEL
LIN {X 0,Y 206.75,Z 329.729,A -85,B 0,C 180,E1 -21083.391,E2 -21083.391} C_VEL
LIN {X 0,Y 206.693,Z 329.727,A -85,B 0,C 180,E1 -21088.427,E2 -21088.427} C_VEL
LIN {X 0,Y 206.706,Z 329.791,A -85,B 0,C 180,E1 -21089.259,E2 -21089.259} C_VEL
LIN {X 0,Y 207.69,Z 332.528,A -85,B 0,C 180,E1 -21089.803,E2 -21089.803} C_VEL
LIN {X 0,Y 209.641,Z 334.617,A -85,B 0,C 180,E1 -21090.657,E2 -21090.657} C_VEL
LIN {X 0,Y 210.624,Z 335.532,A -85,B 0,C 180,E1 -21091.067,E2 -21091.067} C_VEL
LIN {X 0,Y 212.588,Z 338.655,A -85,B 0,C 180,E1 -21091.935,E2 -21091.935} C_VEL
LIN {X 0,Y 214.432,Z 340.622,A -85,B 0,C 180,E1 -21092.668,E2 -21092.668} C_VEL
LIN {X 0,Y 217.133,Z 344.312,A -85,B 0,C 180,E1 -21093.741,E2 -21093.741} C_VEL
LIN {X 0,Y 223.166,Z 353.005,A -85,B 0,C 180,E1 -21095.982,E2 -21095.982} C_VEL
LIN {X 0,Y 229.949,Z 364.695,A -85,B 0,C 180,E1 -21098.341,E2 -21098.341} C_VEL
LIN {X 0,Y 236.754,Z 377.939,A -85,B 0,C 180,E1 -21100.542,E2 -21100.542} C_VEL
LIN {X 0,Y 240.399,Z 385.959,A -85,B 0,C 180,E1 -21101.673,E2 -21101.673} C_VEL
LIN {X 0,Y 237.689,Z 434.923,A -85,B 0,C 180,E1 -21103.088,E2 -21103.088} C_VEL
LIN {X 0,Y 236.127,Z 448.346,A -85,B 0,C 180,E1 -21103.761,E2 -21103.761} C_VEL
LIN {X 0,Y 233.904,Z 461.568,A -85,B 0,C 180,E1 -21104.776,E2 -21104.776} C_VEL
LIN {X 0,Y 231.4,Z 472.916,A -85,B 0,C 180,E1 -21105.991,E2 -21105.991} C_VEL
LIN {X 0,Y 228.398,Z 484.313,A -85,B 0,C 180,E1 -21107.605,E2 -21107.605} C_VEL
LIN {X 0,Y 224.875,Z 495.219,A -85,B 0,C 180,E1 -21109.57,E2 -21109.57} C_VEL
LIN {X 0,Y 221.364,Z 504.595,A -85,B 0,C 180,E1 -21111.748,E2 -21111.748} C_VEL
LIN {X 0,Y 217.549,Z 513.671,A -85,B 0,C 180,E1 -21114.443,E2 -21114.443} C_VEL
LIN {X 0,Y 214.262,Z 520.897,A -85,B 0,C 180,E1 -21117.232,E2 -21117.232} C_VEL
LIN {X 0,Y 211.411,Z 526.606,A -85,B 0,C 180,E1 -21120.088,E2 -21120.088} C_VEL
LIN {X 0,Y 209.117,Z 531.058,A -85,B 0,C 180,E1 -21123.017,E2 -21123.017} C_VEL
LIN {X 0,Y 207.122,Z 534.721,A -85,B 0,C 180,E1 -21126.372,E2 -21126.372} C_VEL
LIN {X 0,Y 205.533,Z 537.229,A -85,B 0,C 180,E1 -21130.004,E2 -21130.004} C_VEL
LIN {X 0,Y 204.962,Z 537.985,A -85,B 0,C 180,E1 -21132.024,E2 -21132.024} C_VEL
LIN {X 0,Y 204.586,Z 538.332,A -85,B 0,C 180,E1 -21134.128,E2 -21134.128} C_VEL
LIN {X 0,Y 204.311,Z 538.278,A -85,B 0,C 180,E1 -21136.066,E2 -21136.066} C_VEL
LIN {X 0,Y 204.132,Z 537.831,A -85,B 0,C 180,E1 -21138.077,E2 -21138.077} C_VEL
LIN {X 0,Y 204.11,Z 536.938,A -85,B 0,C 180,E1 -21140.085,E2 -21140.085} C_VEL
LIN {X 0,Y 204.231,Z 535.643,A -85,B 0,C 180,E1 -21142.087,E2 -21142.087} C_VEL
LIN {X 0,Y 204.618,Z 533.076,A -85,B 0,C 180,E1 -21144.92,E2 -21144.92} C_VEL
LIN {X 0,Y 205.143,Z 529.171,A -85,B 0,C 180,E1 -21148.035,E2 -21148.035} C_VEL
LIN {X 0,Y 205.995,Z 524.313,A -85,B 0,C 180,E1 -21150.976,E2 -21150.976} C_VEL
LIN {X 0,Y 207.167,Z 518.199,A -85,B 0,C 180,E1 -21153.889,E2 -21153.889} C_VEL
LIN {X 0,Y 208.929,Z 510.583,A -85,B 0,C 180,E1 -21156.76,E2 -21156.76} C_VEL
LIN {X 0,Y 210.522,Z 502.813,A -85,B 0,C 180,E1 -21159.123,E2 -21159.123} C_VEL
LIN {X 0,Y 212.827,Z 492.226,A -85,B 0,C 180,E1 -21161.668,E2 -21161.668} C_VEL
LIN {X 0,Y 215.113,Z 481.417,A -85,B 0,C 180,E1 -21163.7,E2 -21163.7} C_VEL
LIN {X 0,Y 216.834,Z 470.929,A -85,B 0,C 180,E1 -21165.267,E2 -21165.267} C_VEL
LIN {X 0,Y 218.457,Z 458.35,A -85,B 0,C 180,E1 -21166.708,E2 -21166.708} C_VEL
LIN {X 0,Y 219.729,Z 445.781,A -85,B 0,C 180,E1 -21167.748,E2 -21167.748} C_VEL
LIN {X 0,Y 220.664,Z 432.465,A -85,B 0,C 180,E1 -21168.45,E2 -21168.45} C_VEL
LIN {X 0,Y 223.178,Z 368.035,A -85,B 0,C 180,E1 -21170.449,E2 -21170.449} C_VEL
LIN {X 0,Y 217.196,Z 351.706,A -85,B 0,C 180,E1 -21171.864,E2 -21171.864} C_VEL
LIN {X 0,Y 212.748,Z 341.839,A -85,B 0,C 180,E1 -21172.893,E2 -21172.893} C_VEL
LIN {X 0,Y 207.885,Z 332.838,A -85,B 0,C 180,E1 -21174.011,E2 -21174.011} C_VEL
LIN {X 0,Y 206.847,Z 330.488,A -85,B 0,C 180,E1 -21174.275,E2 -21174.275} C_VEL
LIN {X 0,Y 206.687,Z 329.739,A -85,B 0,C 180,E1 -21174.417,E2 -21174.417} C_VEL
LIN {X 0,Y 206.685,Z 329.738,A -85,B 0,C 180,E1 -21178.426,E2 -21178.426} C_VEL
LIN {X 0,Y 206.693,Z 329.735,A -85,B 0,C 180,E1 -21182.957,E2 -21182.957} C_VEL
LIN {X 0,Y 206.666,Z 329.741,A -85,B 0,C 180,E1 -21187.741,E2 -21187.741} C_VEL
LIN {X 0,Y 206.628,Z 329.74,A -85,B 0,C 180,E1 -21191.557,E2 -21191.557} C_VEL
LIN {X 0,Y 206.626,Z 329.74,A -85,B 0,C 180,E1 -21195.581,E2 -21195.581} C_VEL
LIN {X 0,Y 206.643,Z 329.741,A -85,B 0,C 180,E1 -21199.744,E2 -21199.744} C_VEL
LIN {X 0,Y 206.695,Z 329.72,A -85,B 0,C 180,E1 -21204.687,E2 -21204.687} C_VEL
LIN {X 0,Y 206.69,Z 329.739,A -85,B 0,C 180,E1 -21209.333,E2 -21209.333} C_VEL
LIN {X 0,Y 206.679,Z 329.718,A -85,B 0,C 180,E1 -21213.764,E2 -21213.764} C_VEL
LIN {X 0,Y 206.707,Z 329.736,A -85,B 0,C 180,E1 -21218.037,E2 -21218.037} C_VEL
LIN {X 0,Y 206.797,Z 329.715,A -85,B 0,C 180,E1 -21222.189,E2 -21222.189} C_VEL
LIN {X 0,Y 206.837,Z 329.705,A -85,B 0,C 180,E1 -21226.24,E2 -21226.24} C_VEL
LIN {X 0,Y 207.065,Z 329.692,A -85,B 0,C 180,E1 -21230.229,E2 -21230.229} C_VEL
LIN {X 0,Y 207.028,Z 329.676,A -85,B 0,C 180,E1 -21234.154,E2 -21234.154} C_VEL
LIN {X 0,Y 207.338,Z 329.649,A -85,B 0,C 180,E1 -21238.057,E2 -21238.057} C_VEL
LIN {X 0,Y 207.472,Z 329.64,A -85,B 0,C 180,E1 -21240,E2 -21240} C_VEL
LIN {X 0,Y 207.339,Z 329.656,A -85,B 0,C 180,E1 -21241.942,E2 -21241.942} C_VEL
LIN {X 0,Y 207.123,Z 329.674,A -85,B 0,C 180,E1 -21247.8,E2 -21247.8} C_VEL
LIN {X 0,Y 206.908,Z 329.709,A -85,B 0,C 180,E1 -21251.759,E2 -21251.759} C_VEL
LIN {X 0,Y 206.822,Z 329.702,A -85,B 0,C 180,E1 -21255.774,E2 -21255.774} C_VEL
LIN {X 0,Y 206.742,Z 329.731,A -85,B 0,C 180,E1 -21259.873,E2 -21259.873} C_VEL
LIN {X 0,Y 206.74,Z 329.727,A -85,B 0,C 180,E1 -21264.075,E2 -21264.075} C_VEL
LIN {X 0,Y 206.73,Z 329.726,A -85,B 0,C 180,E1 -21268.421,E2 -21268.421} C_VEL
LIN {X 0,Y 206.692,Z 329.733,A -85,B 0,C 180,E1 -21272.959,E2 -21272.959} C_VEL
LIN {X 0,Y 206.663,Z 329.74,A -85,B 0,C 180,E1 -21277.743,E2 -21277.743} C_VEL
LIN {X 0,Y 206.631,Z 329.734,A -85,B 0,C 180,E1 -21281.562,E2 -21281.562} C_VEL
LIN {X 0,Y 206.627,Z 329.746,A -85,B 0,C 180,E1 -21285.584,E2 -21285.584} C_VEL
LIN {X 0,Y 206.675,Z 329.741,A -85,B 0,C 180,E1 -21290.687,E2 -21290.687} C_VEL
LIN {X 0,Y 206.696,Z 329.739,A -85,B 0,C 180,E1 -21291.152,E2 -21291.152} C_VEL
LIN {X 0,Y 206.718,Z 330.503,A -85,B 0,C 180,E1 -21291.663,E2 -21291.663} C_VEL
LIN {X 0,Y 206.731,Z 334.017,A -85,B 0,C 180,E1 -21293.147,E2 -21293.147} C_VEL
LIN {X 0,Y 206.777,Z 337.679,A -85,B 0,C 180,E1 -21293.944,E2 -21293.944} C_VEL
LIN {X 0,Y 207.021,Z 343.425,A -85,B 0,C 180,E1 -21294.646,E2 -21294.646} C_VEL
LIN {X 0,Y 208.115,Z 351.781,A -85,B 0,C 180,E1 -21295.386,E2 -21295.386} C_VEL
LIN {X 0,Y 209.296,Z 355.82,A -85,B 0,C 180,E1 -21295.749,E2 -21295.749} C_VEL
LIN {X 0,Y 213.548,Z 367.692,A -85,B 0,C 180,E1 -21296.842,E2 -21296.842} C_VEL
LIN {X 0,Y 216.136,Z 391.573,A -85,B 0,C 180,E1 -21298.095,E2 -21298.095} C_VEL
LIN {X 0,Y 214.046,Z 445.525,A -85,B 0,C 180,E1 -21299.852,E2 -21299.852} C_VEL
LIN {X 0,Y 212.833,Z 459.184,A -85,B 0,C 180,E1 -21300.651,E2 -21300.651} C_VEL
LIN {X 0,Y 211.268,Z 471.263,A -85,B 0,C 180,E1 -21301.705,E2 -21301.705} C_VEL
LIN {X 0,Y 209.504,Z 482.673,A -85,B 0,C 180,E1 -21303.074,E2 -21303.074} C_VEL
LIN {X 0,Y 207.259,Z 494.413,A -85,B 0,C 180,E1 -21304.923,E2 -21304.923} C_VEL
LIN {X 0,Y 204.925,Z 504.952,A -85,B 0,C 180,E1 -21307.04,E2 -21307.04} C_VEL
LIN {X 0,Y 202.906,Z 514.358,A -85,B 0,C 180,E1 -21309.444,E2 -21309.444} C_VEL
LIN {X 0,Y 201.395,Z 521.524,A -85,B 0,C 180,E1 -21311.697,E2 -21311.697} C_VEL
LIN {X 0,Y 199.685,Z 529.249,A -85,B 0,C 180,E1 -21314.696,E2 -21314.696} C_VEL
LIN {X 0,Y 198.485,Z 535.448,A -85,B 0,C 180,E1 -21317.736,E2 -21317.736} C_VEL
LIN {X 0,Y 197.763,Z 540.356,A -85,B 0,C 180,E1 -21320.799,E2 -21320.799} C_VEL
LIN {X 0,Y 197.344,Z 544.112,A -85,B 0,C 180,E1 -21323.868,E2 -21323.868} C_VEL
LIN {X 0,Y 197.245,Z 546.189,A -85,B 0,C 180,E1 -21326.081,E2 -21326.081} C_VEL
LIN {X 0,Y 197.286,Z 547.543,A -85,B 0,C 180,E1 -21327.96,E2 -21327.96} C_VEL
LIN {X 0,Y 197.415,Z 548.587,A -85,B 0,C 180,E1 -21330.001,E2 -21330.001} C_VEL
LIN {X 0,Y 197.247,Z 549.468,A -85,B 0,C 180,E1 -21333.927,E2 -21333.927} C_VEL
LIN {X 0,Y 197.346,Z 549.344,A -85,B 0,C 180,E1 -21336.134,E2 -21336.134} C_VEL
LIN {X 0,Y 198.084,Z 547.838,A -85,B 0,C 180,E1 -21340.22,E2 -21340.22} C_VEL
LIN {X 0,Y 199.624,Z 544.77,A -85,B 0,C 180,E1 -21344.269,E2 -21344.269} C_VEL
LIN {X 0,Y 201.448,Z 541.316,A -85,B 0,C 180,E1 -21347.251,E2 -21347.251} C_VEL
LIN {X 0,Y 203.848,Z 536.804,A -85,B 0,C 180,E1 -21350.169,E2 -21350.169} C_VEL
LIN {X 0,Y 207.301,Z 529.82,A -85,B 0,C 180,E1 -21353.562,E2 -21353.562} C_VEL
LIN {X 0,Y 210.532,Z 522.642,A -85,B 0,C 180,E1 -21356.253,E2 -21356.253} C_VEL
LIN {X 0,Y 214.526,Z 513.524,A -85,B 0,C 180,E1 -21358.897,E2 -21358.897} C_VEL
LIN {X 0,Y 218.617,Z 503.004,A -85,B 0,C 180,E1 -21361.225,E2 -21361.225} C_VEL
LIN {X 0,Y 222.224,Z 492.323,A -85,B 0,C 180,E1 -21363.063,E2 -21363.063} C_VEL
LIN {X 0,Y 225.247,Z 481.97,A -85,B 0,C 180,E1 -21364.44,E2 -21364.44} C_VEL
LIN {X 0,Y 228.236,Z 469.544,A -85,B 0,C 180,E1 -21365.673,E2 -21365.673} C_VEL
LIN {X 0,Y 230.463,Z 456.834,A -85,B 0,C 180,E1 -21366.595,E2 -21366.595} C_VEL
LIN {X 0,Y 232.038,Z 444.042,A -85,B 0,C 180,E1 -21367.192,E2 -21367.192} C_VEL
LIN {X 0,Y 234.523,Z 398.412,A -85,B 0,C 180,E1 -21368.549,E2 -21368.549} C_VEL
LIN {X 0,Y 233.724,Z 393.638,A -85,B 0,C 180,E1 -21368.931,E2 -21368.931} C_VEL
LIN {X 0,Y 228.121,Z 380.665,A -85,B 0,C 180,E1 -21370.846,E2 -21370.846} C_VEL
LIN {X 0,Y 222.42,Z 369.223,A -85,B 0,C 180,E1 -21372.889,E2 -21372.889} C_VEL
LIN {X 0,Y 216.915,Z 359.434,A -85,B 0,C 180,E1 -21374.986,E2 -21374.986} C_VEL
LIN {X 0,Y 212.093,Z 351.532,A -85,B 0,C 180,E1 -21376.966,E2 -21376.966} C_VEL
LIN {X 0,Y 208.533,Z 346.09,A -85,B 0,C 180,E1 -21378.526,E2 -21378.526} C_VEL
LIN {X 0,Y 204.79,Z 340.608,A -85,B 0,C 180,E1 -21380.279,E2 -21380.279} C_VEL
LIN {X 0,Y 201.318,Z 335.689,A -85,B 0,C 180,E1 -21382.027,E2 -21382.027} C_VEL
LIN {X 0,Y 200.976,Z 334.994,A -85,B 0,C 180,E1 -21382.269,E2 -21382.269} C_VEL
LIN {X 0,Y 200.198,Z 332.544,A -85,B 0,C 180,E1 -21384.344,E2 -21384.344} C_VEL
LIN {X 0,Y 199.63,Z 330.618,A -85,B 0,C 180,E1 -21386.251,E2 -21386.251} C_VEL
LIN {X 0,Y 199.688,Z 330.602,A -85,B 0,C 180,E1 -21388.135,E2 -21388.135} C_VEL
LIN {X 0,Y 199.646,Z 330.613,A -85,B 0,C 180,E1 -21392.766,E2 -21392.766} C_VEL
LIN {X 0,Y 199.71,Z 330.61,A -85,B 0,C 180,E1 -21397.226,E2 -21397.226} C_VEL
LIN {X 0,Y 199.752,Z 330.599,A -85,B 0,C 180,E1 -21401.8,E2 -21401.8} C_VEL
LIN {X 0,Y 199.816,Z 330.59,A -85,B 0,C 180,E1 -21405.747,E2 -21405.747} C_VEL
LIN {X 0,Y 200.026,Z 330.563,A -85,B 0,C 180,E1 -21409.882,E2 -21409.882} C_VEL
LIN {X 0,Y 200.016,Z 330.565,A -85,B 0,C 180,E1 -21413.949,E2 -21413.949} C_VEL
LIN {X 0,Y 200.295,Z 330.529,A -85,B 0,C 180,E1 -21417.99,E2 -21417.99} C_VEL
LIN {X 0,Y 200.47,Z 330.497,A -85,B 0,C 180,E1 -21420,E2 -21420} C_VEL
LIN {X 0,Y 200.014,Z 330.557,A -85,B 0,C 180,E1 -21424.03,E2 -21424.03} C_VEL
LIN {X 0,Y 200.082,Z 330.553,A -85,B 0,C 180,E1 -21428.077,E2 -21428.077} C_VEL
LIN {X 0,Y 199.874,Z 330.582,A -85,B 0,C 180,E1 -21432.18,E2 -21432.18} C_VEL
LIN {X 0,Y 199.793,Z 330.592,A -85,B 0,C 180,E1 -21436.345,E2 -21436.345} C_VEL
LIN {X 0,Y 199.679,Z 330.603,A -85,B 0,C 180,E1 -21440.608,E2 -21440.608} C_VEL
LIN {X 0,Y 199.656,Z 330.603,A -85,B 0,C 180,E1 -21444.987,E2 -21444.987} C_VEL
LIN {X 0,Y 199.688,Z 330.604,A -85,B 0,C 180,E1 -21446.311,E2 -21446.311} C_VEL
LIN {X 0,Y 200.531,Z 333.242,A -85,B 0,C 180,E1 -21446.893,E2 -21446.893} C_VEL
LIN {X 0,Y 202.555,Z 335.482,A -85,B 0,C 180,E1 -21447.915,E2 -21447.915} C_VEL
LIN {X 0,Y 203.728,Z 336.344,A -85,B 0,C 180,E1 -21448.459,E2 -21448.459} C_VEL
LIN {X 0,Y 205.534,Z 339.415,A -85,B 0,C 180,E1 -21449.372,E2 -21449.372} C_VEL
LIN {X 0,Y 207.626,Z 341.538,A -85,B 0,C 180,E1 -21450.303,E2 -21450.303} C_VEL
LIN {X 0,Y 210.182,Z 345.127,A -85,B 0,C 180,E1 -21451.444,E2 -21451.444} C_VEL
LIN {X 0,Y 211.848,Z 347.299,A -85,B 0,C 180,E1 -21452.148,E2 -21452.148} C_VEL
LIN {X 0,Y 215.478,Z 352.401,A -85,B 0,C 180,E1 -21453.627,E2 -21453.627} C_VEL
LIN {X 0,Y 219.463,Z 358.165,A -85,B 0,C 180,E1 -21455.153,E2 -21455.153} C_VEL
LIN {X 0,Y 226.076,Z 369.845,A -85,B 0,C 180,E1 -21457.564,E2 -21457.564} C_VEL
LIN {X 0,Y 232.299,Z 382.252,A -85,B 0,C 180,E1 -21459.682,E2 -21459.682} C_VEL
LIN {X 0,Y 235.023,Z 388.366,A -85,B 0,C 180,E1 -21460.576,E2 -21460.576} C_VEL
LIN {X 0,Y 232.336,Z 435.355,A -85,B 0,C 180,E1 -21461.965,E2 -21461.965} C_VEL
LIN {X 0,Y 230.646,Z 449.081,A -85,B 0,C 180,E1 -21462.667,E2 -21462.667} C_VEL
LIN {X 0,Y 228.377,Z 461.982,A -85,B 0,C 180,E1 -21463.681,E2 -21463.681} C_VEL
LIN {X 0,Y 225.772,Z 473.278,A -85,B 0,C 180,E1 -21464.912,E2 -21464.912} C_VEL
LIN {X 0,Y 222.644,Z 484.664,A -85,B 0,C 180,E1 -21466.555,E2 -21466.555} C_VEL
LIN {X 0,Y 218.972,Z 495.521,A -85,B 0,C 180,E1 -21468.549,E2 -21468.549} C_VEL
LIN {X 0,Y 214.944,Z 505.709,A -85,B 0,C 180,E1 -21470.992,E2 -21470.992} C_VEL
LIN {X 0,Y 211.653,Z 513.248,A -85,B 0,C 180,E1 -21473.294,E2 -21473.294} C_VEL
LIN {X 0,Y 208.094,Z 520.614,A -85,B 0,C 180,E1 -21476.132,E2 -21476.132} C_VEL
LIN {X 0,Y 205.082,Z 526.433,A -85,B 0,C 180,E1 -21479.065,E2 -21479.065} C_VEL
LIN {X 0,Y 202.585,Z 530.97,A -85,B 0,C 180,E1 -21482.072,E2 -21482.072} C_VEL
LIN {X 0,Y 200.237,Z 535.005,A -85,B 0,C 180,E1 -21485.863,E2 -21485.863} C_VEL
LIN {X 0,Y 198.664,Z 537.301,A -85,B 0,C 180,E1 -21489.281,E2 -21489.281} C_VEL
LIN {X 0,Y 198.025,Z 538.131,A -85,B 0,C 180,E1 -21491.371,E2 -21491.371} C_VEL
LIN {X 0,Y 197.543,Z 538.537,A -85,B 0,C 180,E1 -21493.861,E2 -21493.861} C_VEL
LIN {X 0,Y 197.073,Z 538.096,A -85,B 0,C 180,E1 -21497.643,E2 -21497.643} C_VEL
LIN {X 0,Y 197.024,Z 537.269,A -85,B 0,C 180,E1 -21499.725,E2 -21499.725} C_VEL
LIN {X 0,Y 197.108,Z 536.012,A -85,B 0,C 180,E1 -21501.799,E2 -21501.799} C_VEL
LIN {X 0,Y 197.531,Z 533.22,A -85,B 0,C 180,E1 -21505.024,E2 -21505.024} C_VEL
LIN {X 0,Y 198.046,Z 529.695,A -85,B 0,C 180,E1 -21507.965,E2 -21507.965} C_VEL
LIN {X 0,Y 198.894,Z 524.926,A -85,B 0,C 180,E1 -21511.011,E2 -21511.011} C_VEL
LIN {X 0,Y 200.344,Z 517.791,A -85,B 0,C 180,E1 -21514.525,E2 -21514.525} C_VEL
LIN {X 0,Y 202.203,Z 509.989,A -85,B 0,C 180,E1 -21517.488,E2 -21517.488} C_VEL
LIN {X 0,Y 204.332,Z 500.266,A -85,B 0,C 180,E1 -21520.402,E2 -21520.402} C_VEL
LIN {X 0,Y 206.382,Z 491.261,A -85,B 0,C 180,E1 -21522.537,E2 -21522.537} C_VEL
LIN {X 0,Y 208.763,Z 480.1,A -85,B 0,C 180,E1 -21524.623,E2 -21524.623} C_VEL
LIN {X 0,Y 210.544,Z 469.225,A -85,B 0,C 180,E1 -21526.232,E2 -21526.232} C_VEL
LIN {X 0,Y 212.132,Z 457.234,A -85,B 0,C 180,E1 -21527.595,E2 -21527.595} C_VEL
LIN {X 0,Y 213.395,Z 444.912,A -85,B 0,C 180,E1 -21528.604,E2 -21528.604} C_VEL
LIN {X 0,Y 214.31,Z 431.796,A -85,B 0,C 180,E1 -21529.281,E2 -21529.281} C_VEL
LIN {X 0,Y 216.812,Z 369.572,A -85,B 0,C 180,E1 -21531.257,E2 -21531.257} C_VEL
LIN {X 0,Y 210.61,Z 352.746,A -85,B 0,C 180,E1 -21532.801,E2 -21532.801} C_VEL
LIN {X 0,Y 205.927,Z 342.818,A -85,B 0,C 180,E1 -21533.934,E2 -21533.934} C_VEL
LIN {X 0,Y 199.987,Z 332.024,A -85,B 0,C 180,E1 -21535.389,E2 -21535.389} C_VEL
LIN {X 0,Y 199.657,Z 330.616,A -85,B 0,C 180,E1 -21535.543,E2 -21535.543} C_VEL
LIN {X 0,Y 199.606,Z 330.62,A -85,B 0,C 180,E1 -21539.531,E2 -21539.531} C_VEL
LIN {X 0,Y 199.664,Z 330.612,A -85,B 0,C 180,E1 -21542.35,E2 -21542.35} C_VEL
LIN {X 0,Y 199.615,Z 330.618,A -85,B 0,C 180,E1 -21546.762,E2 -21546.762} C_VEL
LIN {X 0,Y 199.592,Z 330.619,A -85,B 0,C 180,E1 -21549.33,E2 -21549.33} C_VEL
LIN {X 0,Y 199.563,Z 330.622,A -85,B 0,C 180,E1 -21552.305,E2 -21552.305} C_VEL
LIN {X 0,Y 199.572,Z 330.62,A -85,B 0,C 180,E1 -21555.226,E2 -21555.226} C_VEL
LIN {X 0,Y 199.566,Z 330.614,A -85,B 0,C 180,E1 -21558.001,E2 -21558.001} C_VEL
LIN {X 0,Y 199.593,Z 330.621,A -85,B 0,C 180,E1 -21560.771,E2 -21560.771} C_VEL
LIN {X 0,Y 199.605,Z 330.604,A -85,B 0,C 180,E1 -21565.711,E2 -21565.711} C_VEL
LIN {X 0,Y 199.68,Z 330.608,A -85,B 0,C 180,E1 -21568.133,E2 -21568.133} C_VEL
LIN {X 0,Y 199.628,Z 330.602,A -85,B 0,C 180,E1 -21572.763,E2 -21572.763} C_VEL
LIN {X 0,Y 199.665,Z 330.607,A -85,B 0,C 180,E1 -21577.22,E2 -21577.22} C_VEL
LIN {X 0,Y 199.739,Z 330.596,A -85,B 0,C 180,E1 -21581.802,E2 -21581.802} C_VEL
LIN {X 0,Y 199.756,Z 330.581,A -85,B 0,C 180,E1 -21585.742,E2 -21585.742} C_VEL
LIN {X 0,Y 200.017,Z 330.57,A -85,B 0,C 180,E1 -21589.881,E2 -21589.881} C_VEL
LIN {X 0,Y 199.992,Z 330.553,A -85,B 0,C 180,E1 -21593.948,E2 -21593.948} C_VEL
LIN {X 0,Y 200.28,Z 330.527,A -85,B 0,C 180,E1 -21597.989,E2 -21597.989} C_VEL
LIN {X 0,Y 200.44,Z 330.516,A -85,B 0,C 180,E1 -21600,E2 -21600} C_VEL
LIN {X 0,Y 199.986,Z 330.559,A -85,B 0,C 180,E1 -21604.03,E2 -21604.03} C_VEL
LIN {X 0,Y 200.07,Z 330.553,A -85,B 0,C 180,E1 -21608.077,E2 -21608.077} C_VEL
LIN {X 0,Y 199.858,Z 330.589,A -85,B 0,C 180,E1 -21612.18,E2 -21612.18} C_VEL
LIN {X 0,Y 199.759,Z 330.583,A -85,B 0,C 180,E1 -21616.347,E2 -21616.347} C_VEL
LIN {X 0,Y 199.666,Z 330.614,A -85,B 0,C 180,E1 -21620.609,E2 -21620.609} C_VEL
LIN {X 0,Y 199.658,Z 330.612,A -85,B 0,C 180,E1 -21624.986,E2 -21624.986} C_VEL
LIN {X 0,Y 199.658,Z 330.611,A -85,B 0,C 180,E1 -21629.525,E2 -21629.525} C_VEL
LIN {X 0,Y 199.665,Z 330.609,A -85,B 0,C 180,E1 -21632.356,E2 -21632.356} C_VEL
LIN {X 0,Y 199.612,Z 330.617,A -85,B 0,C 180,E1 -21636.765,E2 -21636.765} C_VEL
LIN {X 0,Y 199.591,Z 330.624,A -85,B 0,C 180,E1 -21639.332,E2 -21639.332} C_VEL
LIN {X 0,Y 199.564,Z 330.612,A -85,B 0,C 180,E1 -21642.31,E2 -21642.31} C_VEL
LIN {X 0,Y 199.573,Z 330.626,A -85,B 0,C 180,E1 -21645.229,E2 -21645.229} C_VEL
LIN {X 0,Y 199.649,Z 330.731,A -85,B 0,C 180,E1 -21650.521,E2 -21650.521} C_VEL
LIN {X 0,Y 201.174,Z 336.906,A -85,B 0,C 180,E1 -21653.655,E2 -21653.655} C_VEL
LIN {X 0,Y 209.093,Z 355.234,A -85,B 0,C 180,E1 -21655.695,E2 -21655.695} C_VEL
LIN {X 0,Y 209.296,Z 355.82,A -85,B 0,C 180,E1 -21655.749,E2 -21655.749} C_VEL
LIN {X 0,Y 210.265,Z 359.476,A -85,B 0,C 180,E1 -21656.04,E2 -21656.04} C_VEL
LIN {X 0,Y 210.662,Z 363.321,A -85,B 0,C 180,E1 -21656.248,E2 -21656.248} C_VEL
LIN {X 0,Y 210.344,Z 371.222,A -85,B 0,C 180,E1 -21656.504,E2 -21656.504} C_VEL
LIN {X 0,Y 209.275,Z 383.337,A -85,B 0,C 180,E1 -21656.81,E2 -21656.81} C_VEL
LIN {X 0,Y 209.387,Z 387.344,A -85,B 0,C 180,E1 -21656.98,E2 -21656.98} C_VEL
LIN {X 0,Y 209.787,Z 393.549,A -85,B 0,C 180,E1 -21657.277,E2 -21657.277} C_VEL
LIN {X 0,Y 207.664,Z 445.513,A -85,B 0,C 180,E1 -21659.017,E2 -21659.017} C_VEL
LIN {X 0,Y 206.385,Z 459.328,A -85,B 0,C 180,E1 -21659.851,E2 -21659.851} C_VEL
LIN {X 0,Y 204.682,Z 471.87,A -85,B 0,C 180,E1 -21660.99,E2 -21660.99} C_VEL
LIN {X 0,Y 202.852,Z 483.056,A -85,B 0,C 180,E1 -21662.396,E2 -21662.396} C_VEL
LIN {X 0,Y 200.533,Z 494.691,A -85,B 0,C 180,E1 -21664.299,E2 -21664.299} C_VEL
LIN {X 0,Y 198.121,Z 505.149,A -85,B 0,C 180,E1 -21666.482,E2 -21666.482} C_VEL
LIN {X 0,Y 196.015,Z 514.553,A -85,B 0,C 180,E1 -21668.991,E2 -21668.991} C_VEL
LIN {X 0,Y 194.642,Z 520.859,A -85,B 0,C 180,E1 -21671.038,E2 -21671.038} C_VEL
LIN {X 0,Y 192.82,Z 528.697,A -85,B 0,C 180,E1 -21674.137,E2 -21674.137} C_VEL
LIN {X 0,Y 191.501,Z 534.962,A -85,B 0,C 180,E1 -21677.281,E2 -21677.281} C_VEL
LIN {X 0,Y 190.721,Z 539.932,A -85,B 0,C 180,E1 -21680.457,E2 -21680.457} C_VEL
LIN {X 0,Y 190.28,Z 543.746,A -85,B 0,C 180,E1 -21683.64,E2 -21683.64} C_VEL
LIN {X 0,Y 190.141,Z 546.189,A -85,B 0,C 180,E1 -21686.35,E2 -21686.35} C_VEL
LIN {X 0,Y 190.315,Z 548.325,A -85,B 0,C 180,E1 -21690.002,E2 -21690.002} C_VEL
LIN {X 0,Y 190.158,Z 549.234,A -85,B 0,C 180,E1 -21693.727,E2 -21693.727} C_VEL
LIN {X 0,Y 190.283,Z 549.164,A -85,B 0,C 180,E1 -21696.363,E2 -21696.363} C_VEL
LIN {X 0,Y 190.562,Z 548.648,A -85,B 0,C 180,E1 -21698.485,E2 -21698.485} C_VEL
LIN {X 0,Y 191.797,Z 546.421,A -85,B 0,C 180,E1 -21702.702,E2 -21702.702} C_VEL
LIN {X 0,Y 193.29,Z 543.68,A -85,B 0,C 180,E1 -21705.826,E2 -21705.826} C_VEL
LIN {X 0,Y 195.452,Z 539.943,A -85,B 0,C 180,E1 -21708.883,E2 -21708.883} C_VEL
LIN {X 0,Y 198.129,Z 535.113,A -85,B 0,C 180,E1 -21711.868,E2 -21711.868} C_VEL
LIN {X 0,Y 201.806,Z 527.928,A -85,B 0,C 180,E1 -21715.254,E2 -21715.254} C_VEL
LIN {X 0,Y 205.489,Z 520.094,A -85,B 0,C 180,E1 -21718.053,E2 -21718.053} C_VEL
LIN {X 0,Y 209.879,Z 510.351,A -85,B 0,C 180,E1 -21720.709,E2 -21720.709} C_VEL
LIN {X 0,Y 213.889,Z 500.246,A -85,B 0,C 180,E1 -21722.832,E2 -21722.832} C_VEL
LIN {X 0,Y 217.65,Z 488.849,A -85,B 0,C 180,E1 -21724.69,E2 -21724.69} C_VEL
LIN {X 0,Y 220.878,Z 477.65,A -85,B 0,C 180,E1 -21726.062,E2 -21726.062} C_VEL
LIN {X 0,Y 223.727,Z 465.05,A -85,B 0,C 180,E1 -21727.209,E2 -21727.209} C_VEL
LIN {X 0,Y 225.914,Z 451.59,A -85,B 0,C 180,E1 -21728.051,E2 -21728.051} C_VEL
LIN {X 0,Y 227.138,Z 438.561,A -85,B 0,C 180,E1 -21728.571,E2 -21728.571} C_VEL
LIN {X 0,Y 229.319,Z 399.507,A -85,B 0,C 180,E1 -21729.725,E2 -21729.725} C_VEL
LIN {X 0,Y 228.795,Z 396.678,A -85,B 0,C 180,E1 -21729.975,E2 -21729.975} C_VEL
LIN {X 0,Y 223.08,Z 383.317,A -85,B 0,C 180,E1 -21732.05,E2 -21732.05} C_VEL
LIN {X 0,Y 217.222,Z 371.505,A -85,B 0,C 180,E1 -21734.289,E2 -21734.289} C_VEL
LIN {X 0,Y 211.427,Z 361.309,A -85,B 0,C 180,E1 -21736.667,E2 -21736.667} C_VEL
LIN {X 0,Y 208.099,Z 355.963,A -85,B 0,C 180,E1 -21738.126,E2 -21738.126} C_VEL
LIN {X 0,Y 205.193,Z 351.425,A -85,B 0,C 180,E1 -21739.474,E2 -21739.474} C_VEL
LIN {X 0,Y 201.647,Z 346.122,A -85,B 0,C 180,E1 -21741.225,E2 -21741.225} C_VEL
LIN {X 0,Y 197.576,Z 340.312,A -85,B 0,C 180,E1 -21743.409,E2 -21743.409} C_VEL
LIN {X 0,Y 194.077,Z 335.614,A -85,B 0,C 180,E1 -21745.463,E2 -21745.463} C_VEL
LIN {X 0,Y 193.547,Z 334.535,A -85,B 0,C 180,E1 -21745.907,E2 -21745.907} C_VEL
LIN {X 0,Y 192.584,Z 331.49,A -85,B 0,C 180,E1 -21748.972,E2 -21748.972} C_VEL
LIN {X 0,Y 192.623,Z 331.482,A -85,B 0,C 180,E1 -21751.686,E2 -21751.686} C_VEL
LIN {X 0,Y 192.682,Z 331.478,A -85,B 0,C 180,E1 -21756.346,E2 -21756.346} C_VEL
LIN {X 0,Y 192.7,Z 331.479,A -85,B 0,C 180,E1 -21761.489,E2 -21761.489} C_VEL
LIN {X 0,Y 192.742,Z 331.474,A -85,B 0,C 180,E1 -21765.212,E2 -21765.212} C_VEL
LIN {X 0,Y 192.949,Z 331.447,A -85,B 0,C 180,E1 -21769.567,E2 -21769.567} C_VEL
LIN {X 0,Y 193.037,Z 331.422,A -85,B 0,C 180,E1 -21771.627,E2 -21771.627} C_VEL
LIN {X 0,Y 193.24,Z 331.407,A -85,B 0,C 180,E1 -21777.916,E2 -21777.916} C_VEL
LIN {X 0,Y 193.435,Z 331.373,A -85,B 0,C 180,E1 -21780,E2 -21780} C_VEL
LIN {X 0,Y 192.96,Z 331.435,A -85,B 0,C 180,E1 -21784.178,E2 -21784.178} C_VEL
LIN {X 0,Y 193.032,Z 331.429,A -85,B 0,C 180,E1 -21788.374,E2 -21788.374} C_VEL
LIN {X 0,Y 192.801,Z 331.46,A -85,B 0,C 180,E1 -21792.634,E2 -21792.634} C_VEL
LIN {X 0,Y 192.752,Z 331.465,A -85,B 0,C 180,E1 -21796.96,E2 -21796.96} C_VEL
LIN {X 0,Y 192.661,Z 331.477,A -85,B 0,C 180,E1 -21802.522,E2 -21802.522} C_VEL
LIN {X 0,Y 192.704,Z 331.712,A -85,B 0,C 180,E1 -21802.941,E2 -21802.941} C_VEL
LIN {X 0,Y 193.505,Z 334.059,A -85,B 0,C 180,E1 -21803.548,E2 -21803.548} C_VEL
LIN {X 0,Y 195.537,Z 336.382,A -85,B 0,C 180,E1 -21804.76,E2 -21804.76} C_VEL
LIN {X 0,Y 196.917,Z 337.321,A -85,B 0,C 180,E1 -21805.501,E2 -21805.501} C_VEL
LIN {X 0,Y 198.779,Z 340.481,A -85,B 0,C 180,E1 -21806.582,E2 -21806.582} C_VEL
LIN {X 0,Y 201.038,Z 342.616,A -85,B 0,C 180,E1 -21807.719,E2 -21807.719} C_VEL
LIN {X 0,Y 203.278,Z 345.969,A -85,B 0,C 180,E1 -21808.866,E2 -21808.866} C_VEL
LIN {X 0,Y 204.928,Z 347.875,A -85,B 0,C 180,E1 -21809.639,E2 -21809.639} C_VEL
LIN {X 0,Y 207.923,Z 351.726,A -85,B 0,C 180,E1 -21810.997,E2 -21810.997} C_VEL
LIN {X 0,Y 215.601,Z 362.926,A -85,B 0,C 180,E1 -21814.206,E2 -21814.206} C_VEL
LIN {X 0,Y 222.295,Z 375.006,A -85,B 0,C 180,E1 -21816.775,E2 -21816.775} C_VEL
LIN {X 0,Y 228.142,Z 387,A -85,B 0,C 180,E1 -21818.865,E2 -21818.865} C_VEL
LIN {X 0,Y 229.762,Z 390.667,A -85,B 0,C 180,E1 -21819.428,E2 -21819.428} C_VEL
LIN {X 0,Y 227.011,Z 436.296,A -85,B 0,C 180,E1 -21820.808,E2 -21820.808} C_VEL
LIN {X 0,Y 225.327,Z 449.317,A -85,B 0,C 180,E1 -21821.486,E2 -21821.486} C_VEL
LIN {X 0,Y 223.191,Z 461.302,A -85,B 0,C 180,E1 -21822.436,E2 -21822.436} C_VEL
LIN {X 0,Y 220.686,Z 471.992,A -85,B 0,C 180,E1 -21823.571,E2 -21823.571} C_VEL
LIN {X 0,Y 217.692,Z 482.736,A -85,B 0,C 180,E1 -21825.077,E2 -21825.077} C_VEL
LIN {X 0,Y 213.958,Z 493.659,A -85,B 0,C 180,E1 -21827.031,E2 -21827.031} C_VEL
LIN {X 0,Y 210.067,Z 503.466,A -85,B 0,C 180,E1 -21829.276,E2 -21829.276} C_VEL
LIN {X 0,Y 206.71,Z 510.957,A -85,B 0,C 180,E1 -21831.444,E2 -21831.444} C_VEL
LIN {X 0,Y 202.625,Z 519.16,A -85,B 0,C 180,E1 -21834.48,E2 -21834.48} C_VEL
LIN {X 0,Y 198.826,Z 526.249,A -85,B 0,C 180,E1 -21837.979,E2 -21837.979} C_VEL
LIN {X 0,Y 196.112,Z 530.883,A -85,B 0,C 180,E1 -21841.065,E2 -21841.065} C_VEL
LIN {X 0,Y 193.971,Z 534.369,A -85,B 0,C 180,E1 -21844.227,E2 -21844.227} C_VEL
LIN {X 0,Y 192.814,Z 536.082,A -85,B 0,C 180,E1 -21846.361,E2 -21846.361} C_VEL
LIN {X 0,Y 191.832,Z 537.375,A -85,B 0,C 180,E1 -21848.507,E2 -21848.507} C_VEL
LIN {X 0,Y 191.108,Z 538.26,A -85,B 0,C 180,E1 -21850.671,E2 -21850.671} C_VEL
LIN {X 0,Y 190.487,Z 538.744,A -85,B 0,C 180,E1 -21853.593,E2 -21853.593} C_VEL
LIN {X 0,Y 189.999,Z 538.354,A -85,B 0,C 180,E1 -21857.176,E2 -21857.176} C_VEL
LIN {X 0,Y 189.935,Z 537.591,A -85,B 0,C 180,E1 -21859.337,E2 -21859.337} C_VEL
LIN {X 0,Y 189.979,Z 536.381,A -85,B 0,C 180,E1 -21861.489,E2 -21861.489} C_VEL
LIN {X 0,Y 190.443,Z 533.359,A -85,B 0,C 180,E1 -21865.139,E2 -21865.139} C_VEL
LIN {X 0,Y 190.947,Z 530.218,A -85,B 0,C 180,E1 -21867.889,E2 -21867.889} C_VEL
LIN {X 0,Y 191.792,Z 525.536,A -85,B 0,C 180,E1 -21871.048,E2 -21871.048} C_VEL
LIN {X 0,Y 193.265,Z 518.496,A -85,B 0,C 180,E1 -21874.692,E2 -21874.692} C_VEL
LIN {X 0,Y 195.18,Z 510.853,A -85,B 0,C 180,E1 -21877.759,E2 -21877.759} C_VEL
LIN {X 0,Y 197.358,Z 501.269,A -85,B 0,C 180,E1 -21880.773,E2 -21880.773} C_VEL
LIN {X 0,Y 199.717,Z 491.354,A -85,B 0,C 180,E1 -21883.221,E2 -21883.221} C_VEL
LIN {X 0,Y 201.932,Z 481.565,A -85,B 0,C 180,E1 -21885.129,E2 -21885.129} C_VEL
LIN {X 0,Y 204.061,Z 469.243,A -85,B 0,C 180,E1 -21887.021,E2 -21887.021} C_VEL
LIN {X 0,Y 205.719,Z 457.199,A -85,B 0,C 180,E1 -21888.42,E2 -21888.42} C_VEL
LIN {X 0,Y 207.037,Z 444.737,A -85,B 0,C 180,E1 -21889.455,E2 -21889.455} C_VEL
LIN {X 0,Y 208.002,Z 431.072,A -85,B 0,C 180,E1 -21890.161,E2 -21890.161} C_VEL
LIN {X 0,Y 210.526,Z 371.134,A -85,B 0,C 180,E1 -21892.107,E2 -21892.107} C_VEL
LIN {X 0,Y 204.244,Z 354.317,A -85,B 0,C 180,E1 -21893.75,E2 -21893.75} C_VEL
LIN {X 0,Y 198.992,Z 343.814,A -85,B 0,C 180,E1 -21895.074,E2 -21895.074} C_VEL
LIN {X 0,Y 194.06,Z 334.946,A -85,B 0,C 180,E1 -21896.357,E2 -21896.357} C_VEL
LIN {X 0,Y 192.737,Z 332.28,A -85,B 0,C 180,E1 -21896.728,E2 -21896.728} C_VEL
LIN {X 0,Y 192.614,Z 331.492,A -85,B 0,C 180,E1 -21896.873,E2 -21896.873} C_VEL
LIN {X 0,Y 192.569,Z 331.495,A -85,B 0,C 180,E1 -21900.725,E2 -21900.725} C_VEL
LIN {X 0,Y 192.593,Z 331.491,A -85,B 0,C 180,E1 -21903.185,E2 -21903.185} C_VEL
LIN {X 0,Y 192.539,Z 331.503,A -85,B 0,C 180,E1 -21908.352,E2 -21908.352} C_VEL
LIN {X 0,Y 192.482,Z 331.509,A -85,B 0,C 180,E1 -21913.092,E2 -21913.092} C_VEL
LIN {X 0,Y 192.48,Z 331.494,A -85,B 0,C 180,E1 -21916.905,E2 -21916.905} C_VEL
LIN {X 0,Y 192.537,Z 331.497,A -85,B 0,C 180,E1 -21921.644,E2 -21921.644} C_VEL
LIN {X 0,Y 192.59,Z 331.483,A -85,B 0,C 180,E1 -21926.812,E2 -21926.812} C_VEL
LIN {X 0,Y 192.613,Z 331.482,A -85,B 0,C 180,E1 -21931.683,E2 -21931.683} C_VEL
LIN {X 0,Y 192.652,Z 331.477,A -85,B 0,C 180,E1 -21936.341,E2 -21936.341} C_VEL
LIN {X 0,Y 192.688,Z 331.477,A -85,B 0,C 180,E1 -21941.491,E2 -21941.491} C_VEL
LIN {X 0,Y 192.692,Z 331.457,A -85,B 0,C 180,E1 -21945.208,E2 -21945.208} C_VEL
LIN {X 0,Y 192.939,Z 331.45,A -85,B 0,C 180,E1 -21949.566,E2 -21949.566} C_VEL
LIN {X 0,Y 192.955,Z 331.431,A -85,B 0,C 180,E1 -21953.726,E2 -21953.726} C_VEL
LIN {X 0,Y 193.224,Z 331.405,A -85,B 0,C 180,E1 -21957.915,E2 -21957.915} C_VEL
LIN {X 0,Y 193.406,Z 331.392,A -85,B 0,C 180,E1 -21960,E2 -21960} C_VEL
LIN {X 0,Y 192.933,Z 331.435,A -85,B 0,C 180,E1 -21964.178,E2 -21964.178} C_VEL
LIN {X 0,Y 193.02,Z 331.432,A -85,B 0,C 180,E1 -21968.374,E2 -21968.374} C_VEL
LIN {X 0,Y 192.784,Z 331.466,A -85,B 0,C 180,E1 -21972.634,E2 -21972.634} C_VEL
LIN {X 0,Y 192.713,Z 331.463,A -85,B 0,C 180,E1 -21976.962,E2 -21976.962} C_VEL
LIN {X 0,Y 192.603,Z 331.491,A -85,B 0,C 180,E1 -21981.401,E2 -21981.401} C_VEL
LIN {X 0,Y 192.641,Z 331.483,A -85,B 0,C 180,E1 -21984.213,E2 -21984.213} C_VEL
